C07281=1048.225,401.542,372.791,174.335,42.188,158.264
C07282=1048.234,401.788,372.747,174.343,42.195,158.266
C07283=1048.243,402.034,372.703,174.350,42.201,158.268
C07284=1048.252,402.280,372.659,174.359,42.208,158.271
C07285=1048.261,402.526,372.615,174.367,42.215,158.273
C07286=1048.270,402.772,372.571,174.375,42.222,158.275
C07287=1048.279,403.018,372.526,174.384,42.229,158.278
C07288=1048.288,403.264,372.482,174.391,42.236,158.280
C07289=1048.298,403.509,372.437,174.399,42.243,158.282
C07290=1048.311,403.897,372.367,174.413,42.254,158.286
C07291=1048.326,404.285,372.298,174.425,42.265,158.290
C07292=1048.340,404.673,372.227,174.439,42.276,158.294
C07293=1048.354,405.061,372.157,174.452,42.288,158.297
C07294=1048.363,405.308,372.113,174.461,42.295,158.300
C07295=1048.372,405.553,372.068,174.468,42.302,158.302
C07296=1048.381,405.799,372.022,174.478,42.309,158.305
C07297=1048.390,406.044,371.979,174.485,42.316,158.307
C07298=1048.399,406.290,371.933,174.495,42.324,158.310
C07299=1048.409,406.536,371.889,174.502,42.331,158.312
C07300=1048.417,406.782,371.844,174.511,42.338,158.314
C07301=1048.427,407.028,371.799,174.519,42.345,158.317
C07302=1048.436,407.274,371.754,174.528,42.353,158.319
C07303=1048.446,407.520,371.709,174.537,42.360,158.322
C07304=1048.455,407.765,371.664,174.545,42.367,158.324
C07305=1048.464,408.011,371.619,174.555,42.374,158.327
C07306=1048.473,408.257,371.574,174.563,42.382,158.329
C07307=1048.483,408.502,371.529,174.572,42.389,158.332
C07308=1048.492,408.748,371.483,174.580,42.397,158.334
C07309=1048.502,408.994,371.439,174.589,42.404,158.337
C07310=1048.511,409.239,371.393,174.598,42.412,158.339
C07311=1048.520,409.485,371.348,174.606,42.419,158.342
C07312=1048.529,409.731,371.303,174.615,42.427,158.344
C07313=1048.539,409.976,371.258,174.625,42.434,158.347
C07314=1048.548,410.222,371.213,174.633,42.442,158.350
C07315=1048.557,410.468,371.167,174.642,42.449,158.352
C07316=1048.567,410.714,371.122,174.651,42.456,158.355
C07317=1048.577,410.959,371.076,174.660,42.464,158.357
C07318=1048.586,411.205,371.031,174.669,42.472,158.360
C07319=1048.595,411.451,370.986,174.678,42.479,158.362
C07320=1048.606,411.696,370.940,174.687,42.487,158.365
C07321=1048.615,411.942,370.894,174.696,42.495,158.368
C07322=1048.624,412.187,370.848,174.705,42.502,158.370
C07323=1048.635,412.433,370.803,174.715,42.510,158.373
C07324=1048.643,412.679,370.758,174.724,42.518,158.376
C07325=1048.653,412.925,370.712,174.732,42.526,158.378
C07326=1048.663,413.170,370.665,174.742,42.534,158.381
C07327=1048.672,413.416,370.620,174.751,42.541,158.384
C07328=1048.682,413.662,370.574,174.761,42.549,158.387
C07329=1048.692,413.907,370.528,174.770,42.557,158.389
C07330=1048.701,414.152,370.481,174.779,42.565,158.392
C07331=1048.711,414.398,370.435,174.789,42.573,158.395
C07332=1048.720,414.643,370.389,174.798,42.581,158.397
C07333=1048.730,414.889,370.342,174.807,42.589,158.400
C07334=1048.739,415.134,370.296,174.817,42.597,158.403
C07335=1048.749,415.380,370.250,174.826,42.604,158.406
C07336=1048.758,415.626,370.204,174.836,42.613,158.409
C07337=1048.769,415.871,370.158,174.845,42.621,158.411
C07338=1048.778,416.116,370.111,174.855,42.629,158.414
C07339=1048.788,416.362,370.065,174.864,42.637,158.417
C07340=1048.797,416.607,370.019,174.874,42.645,158.420
C07341=1048.808,416.853,369.972,174.883,42.653,158.423
C07342=1048.817,417.099,369.925,174.893,42.662,158.425
C07343=1048.827,417.344,369.879,174.903,42.669,158.428
C07344=1048.837,417.589,369.832,174.913,42.678,158.431
C07345=1048.847,417.835,369.785,174.923,42.686,158.434
C07346=1048.862,418.230,369.710,174.939,42.699,158.439
C07347=1048.879,418.625,369.635,174.954,42.712,158.443
C07348=1048.895,419.020,369.559,174.970,42.726,158.448
C07349=1048.911,419.415,369.483,174.986,42.740,158.453
C07350=1048.921,419.660,369.437,174.996,42.748,158.456
C07351=1048.930,419.906,369.389,175.007,42.756,158.459
C07352=1048.940,420.152,369.342,175.017,42.765,158.462
C07353=1048.950,420.397,369.295,175.026,42.774,158.465
C07354=1048.960,420.642,369.248,175.037,42.782,158.468
C07355=1048.971,420.887,369.201,175.047,42.791,158.471
C07356=1048.980,421.133,369.153,175.058,42.799,158.474
C07357=1048.990,421.378,369.106,175.068,42.808,158.477
C07358=1049.001,421.623,369.058,175.078,42.816,158.480
C07359=1049.011,421.868,369.010,175.088,42.825,158.483
C07360=1049.020,422.114,368.963,175.098,42.834,158.486
C07361=1049.031,422.359,368.915,175.109,42.842,158.489
C07362=1049.041,422.604,368.868,175.119,42.851,158.492
C07363=1049.051,422.849,368.820,175.130,42.860,158.495
C07364=1049.061,423.094,368.773,175.141,42.868,158.499
C07365=1049.071,423.339,368.725,175.151,42.878,158.502
C07366=1049.082,423.585,368.677,175.162,42.886,158.505
C07367=1049.093,423.830,368.629,175.172,42.895,158.508
C07368=1049.103,424.075,368.582,175.183,42.904,158.511
C07369=1049.112,424.320,368.533,175.194,42.913,158.514
C07370=1049.123,424.566,368.486,175.204,42.922,158.518
C07371=1049.134,424.811,368.438,175.215,42.931,158.521
C07372=1049.144,425.056,368.389,175.226,42.939,158.524
C07373=1049.154,425.302,368.342,175.236,42.949,158.527
C07374=1049.165,425.546,368.294,175.247,42.957,158.530
C07375=1049.175,425.792,368.245,175.259,42.966,158.534
C07376=1049.186,426.037,368.197,175.270,42.976,158.537
C07377=1049.195,426.282,368.148,175.280,42.985,158.540
C07378=1049.207,426.527,368.100,175.291,42.994,158.544
C07379=1049.216,426.772,368.052,175.303,43.003,158.547
C07380=1049.227,427.017,368.003,175.314,43.012,158.550
C07381=1049.237,427.262,367.954,175.325,43.021,158.554
C07382=1049.249,427.507,367.906,175.336,43.031,158.557
C07383=1049.258,427.752,367.857,175.348,43.040,158.560
C07384=1049.269,427.997,367.809,175.359,43.049,158.564
C07385=1049.279,428.242,367.760,175.369,43.059,158.567
C07386=1049.291,428.487,367.711,175.381,43.068,158.571
C07387=1049.301,428.732,367.662,175.392,43.078,158.574
C07388=1049.311,428.977,367.613,175.403,43.087,158.577
C07389=1049.322,429.222,367.564,175.416,43.096,158.581
C07390=1049.332,429.467,367.516,175.427,43.106,158.584
C07391=1049.344,429.712,367.467,175.439,43.116,158.588
C07392=1049.354,429.957,367.417,175.450,43.125,158.591
C07393=1049.365,430.202,367.367,175.462,43.135,158.595
C07394=1049.375,430.447,367.319,175.473,43.144,158.599
C07395=1049.385,430.692,367.269,175.485,43.154,158.602
C07396=1049.397,430.937,367.220,175.496,43.163,158.606
C07397=1049.407,431.182,367.171,175.508,43.173,158.609
C07398=1049.417,431.426,367.121,175.521,43.183,158.613
C07399=1049.428,431.671,367.072,175.532,43.193,158.616
C07400=1049.440,431.915,367.022,175.544,43.203,158.620
C07401=1049.451,432.160,366.973,175.557,43.212,158.624
C07402=1049.459,432.370,366.930,175.567,43.221,158.627
C07403=1049.469,432.579,366.888,175.577,43.229,158.630
C07404=1049.478,432.788,366.845,175.587,43.237,158.633
C07405=1049.487,432.997,366.803,175.598,43.246,158.636
C07406=1049.498,433.207,366.760,175.608,43.254,158.639
C07407=1049.507,433.416,366.717,175.618,43.263,158.642
C07408=1049.516,433.625,366.675,175.629,43.271,158.646
C07409=1049.525,433.834,366.632,175.639,43.280,158.649
C07410=1049.536,434.079,366.583,175.651,43.290,158.653
C07411=1049.547,434.323,366.533,175.664,43.300,158.656
C07412=1049.559,434.569,366.482,175.676,43.310,158.660
C07413=1049.570,434.813,366.432,175.689,43.320,158.664
C07414=1049.581,435.058,366.382,175.702,43.330,158.668
C07415=1049.592,435.302,366.332,175.714,43.341,158.672
C07416=1049.604,435.547,366.282,175.726,43.351,158.675
C07417=1049.615,435.792,366.231,175.739,43.361,158.679
C07418=1049.626,436.036,366.181,175.752,43.371,158.683
C07419=1049.637,436.281,366.130,175.764,43.381,158.687
C07420=1049.648,436.526,366.080,175.778,43.391,158.691
C07421=1049.659,436.770,366.030,175.790,43.402,158.695
C07422=1049.671,437.015,365.979,175.803,43.412,158.699
C07423=1049.682,437.259,365.928,175.816,43.423,158.703
C07424=1049.694,437.504,365.877,175.829,43.433,158.707
C07425=1049.705,437.749,365.827,175.841,43.444,158.711
C07426=1049.717,437.993,365.776,175.855,43.455,158.715
C07427=1049.728,438.238,365.725,175.868,43.465,158.719
C07428=1049.740,438.482,365.674,175.881,43.476,158.723
C07429=1049.750,438.727,365.624,175.894,43.486,158.727
C07430=1049.762,438.971,365.572,175.908,43.497,158.731
C07431=1049.774,439.216,365.520,175.921,43.508,158.735
C07432=1049.785,439.460,365.469,175.935,43.518,158.739
C07433=1049.797,439.704,365.418,175.948,43.529,158.743
C07434=1049.808,439.949,365.367,175.961,43.540,158.747
C07435=1049.820,440.193,365.316,175.975,43.551,158.751
C07436=1049.831,440.438,365.264,175.988,43.562,158.756
C07437=1049.843,440.682,365.212,176.002,43.573,158.760
C07438=1049.855,440.926,365.160,176.016,43.583,158.764
C07439=1049.866,441.170,365.109,176.030,43.594,158.768
C07440=1049.878,441.415,365.058,176.043,43.605,158.772
C07441=1049.890,441.659,365.007,176.057,43.616,158.777
C07442=1049.901,441.903,364.954,176.072,43.627,158.781
C07443=1049.913,442.148,364.902,176.085,43.639,158.785
C07444=1049.925,442.392,364.850,176.099,43.650,158.790
C07445=1049.936,442.637,364.798,176.114,43.661,158.794
C07446=1049.949,442.880,364.746,176.128,43.672,158.798
C07447=1049.961,443.124,364.694,176.141,43.683,158.803
C07448=1049.973,443.369,364.643,176.156,43.695,158.807
C07449=1049.984,443.613,364.590,176.170,43.706,158.812
C07450=1049.996,443.857,364.538,176.185,43.717,158.816
C07451=1050.009,444.101,364.486,176.199,43.729,158.821
C07452=1050.020,444.345,364.433,176.214,43.740,158.825
C07453=1050.033,444.590,364.381,176.229,43.752,158.830
C07454=1050.045,444.834,364.328,176.243,43.763,158.834
C07455=1050.056,445.078,364.276,176.258,43.775,158.839
C07456=1050.069,445.322,364.223,176.273,43.786,158.843
C07457=1050.081,445.566,364.171,176.287,43.798,158.848
C07458=1050.093,445.809,364.119,176.302,43.809,158.852
C07459=1050.106,446.052,364.066,176.317,43.821,158.857
C07460=1050.119,446.296,364.014,176.332,43.832,158.862
C07461=1050.132,446.540,363.962,176.347,43.843,158.866
C07462=1050.148,446.805,363.907,176.364,43.856,158.871
C07463=1050.165,447.073,363.851,176.380,43.868,158.876
C07464=1050.182,447.340,363.797,176.396,43.879,158.881
C07465=1050.201,447.608,363.743,176.414,43.891,158.886
C07466=1050.219,447.852,363.694,176.430,43.901,158.890
C07467=1050.237,448.096,363.647,176.444,43.912,158.894
C07468=1050.255,448.341,363.599,176.460,43.922,158.899
C07469=1050.275,448.586,363.552,176.476,43.932,158.903
C07470=1050.296,448.830,363.505,176.492,43.942,158.907
C07471=1050.317,449.075,363.459,176.508,43.951,158.911
C07472=1050.338,449.321,363.414,176.523,43.961,158.916
C07473=1050.361,449.566,363.369,176.540,43.971,158.920
C07474=1050.384,449.811,363.325,176.556,43.980,158.924
C07475=1050.408,450.056,363.281,176.572,43.989,158.928
C07476=1050.432,450.302,363.238,176.588,43.998,158.932
C07477=1050.458,450.546,363.195,176.605,44.007,158.936
C07478=1050.144,450.574,362.895,176.604,44.099,158.963
C07479=1050.118,450.329,362.938,176.588,44.090,158.959
C07480=1050.094,450.083,362.981,176.572,44.081,158.955
C07481=1050.070,449.838,363.025,176.556,44.073,158.951
C07482=1050.046,449.593,363.069,176.539,44.064,158.947
C07483=1050.024,449.348,363.113,176.523,44.054,158.942
C07484=1050.002,449.103,363.159,176.507,44.044,158.938
C07485=1049.981,448.858,363.205,176.492,44.034,158.934
C07486=1049.960,448.613,363.251,176.475,44.025,158.930
C07487=1049.941,448.368,363.298,176.460,44.015,158.925
C07488=1049.921,448.124,363.346,176.444,44.005,158.921
C07489=1049.903,447.880,363.393,176.428,43.995,158.917
C07490=1049.886,447.636,363.442,176.412,43.985,158.912
C07491=1049.868,447.386,363.493,176.397,43.973,158.908
C07492=1049.851,447.137,363.543,176.381,43.963,158.903
C07493=1049.836,446.888,363.594,176.365,43.952,158.899
C07494=1049.821,446.639,363.646,176.350,43.940,158.894
C07495=1049.806,446.395,363.697,176.335,43.929,158.890
C07496=1049.792,446.151,363.749,176.320,43.918,158.885
C07497=1049.779,445.908,363.801,176.305,43.907,158.881
C07498=1049.767,445.666,363.853,176.290,43.895,158.876
C07499=1049.755,445.422,363.906,176.275,43.884,158.871
C07500=1049.743,445.177,363.959,176.260,43.872,158.867
C07501=1049.730,444.933,364.011,176.246,43.861,158.862
C07502=1049.719,444.690,364.064,176.231,43.850,158.858
C07503=1049.706,444.446,364.116,176.216,43.838,158.853
C07504=1049.694,444.201,364.169,176.202,43.826,158.849
C07505=1049.682,443.957,364.221,176.187,43.816,158.844
C07506=1049.670,443.713,364.274,176.173,43.804,158.840
C07507=1049.658,443.469,364.325,176.158,43.793,158.835
C07508=1049.647,443.224,364.378,176.144,43.782,158.831
C07509=1049.635,442.980,364.430,176.129,43.770,158.826
C07510=1049.622,442.737,364.482,176.115,43.759,158.822
C07511=1049.611,442.492,364.534,176.101,43.748,158.818
C07512=1049.599,442.248,364.586,176.087,43.737,158.813
C07513=1049.587,442.003,364.637,176.072,43.726,158.809
C07514=1049.575,441.759,364.690,176.059,43.715,158.805
C07515=1049.564,441.515,364.742,176.045,43.704,158.800
C07516=1049.552,441.270,364.793,176.030,43.693,158.796
C07517=1049.540,441.026,364.845,176.017,43.682,158.792
C07518=1049.528,440.782,364.896,176.003,43.672,158.788
C07519=1049.516,440.537,364.948,175.989,43.660,158.783
C07520=1049.504,440.293,364.999,175.976,43.650,158.779
C07521=1049.494,440.049,365.051,175.962,43.639,158.775
C07522=1049.482,439.804,365.102,175.948,43.628,158.771
C07523=1049.470,439.560,365.154,175.935,43.618,158.767
C07524=1049.458,439.316,365.205,175.921,43.607,158.763
C07525=1049.447,439.071,365.256,175.908,43.596,158.759
C07526=1049.435,438.826,365.307,175.894,43.585,158.754
C07527=1049.424,438.582,365.358,175.881,43.575,158.750
C07528=1049.413,438.337,365.410,175.868,43.564,158.746
C07529=1049.401,438.092,365.461,175.855,43.554,158.742
C07530=1049.390,437.849,365.512,175.841,43.543,158.738
C07531=1049.378,437.603,365.562,175.829,43.533,158.734
C07532=1049.367,437.360,365.613,175.816,43.522,158.730
C07533=1049.355,437.114,365.664,175.803,43.512,158.726
C07534=1049.344,436.870,365.714,175.789,43.502,158.722
C07535=1049.333,436.626,365.765,175.776,43.492,158.718
C07536=1049.322,436.381,365.816,175.764,43.481,158.715
C07537=1049.311,436.137,365.866,175.751,43.471,158.711
C07538=1049.299,435.892,365.917,175.738,43.460,158.707
C07539=1049.287,435.647,365.967,175.725,43.451,158.703
C07540=1049.276,435.403,366.017,175.713,43.440,158.699
C07541=1049.265,435.158,366.068,175.700,43.430,158.695
C07542=1049.254,434.913,366.117,175.687,43.420,158.691
C07543=1049.243,434.668,366.168,175.675,43.410,158.688
C07544=1049.231,434.424,366.218,175.662,43.400,158.684
C07545=1049.220,434.180,366.268,175.650,43.390,158.680
C07546=1049.209,433.934,366.318,175.637,43.380,158.676
C07547=1049.200,433.724,366.361,175.627,43.372,158.673
C07548=1049.190,433.514,366.404,175.616,43.363,158.670
C07549=1049.180,433.304,366.446,175.606,43.355,158.667
C07550=1049.171,433.094,366.489,175.596,43.346,158.663
C07551=1049.161,432.884,366.532,175.585,43.338,158.660
C07552=1049.152,432.673,366.575,175.574,43.329,158.657
C07553=1049.143,432.463,366.618,175.563,43.321,158.654
C07554=1049.134,432.253,366.660,175.553,43.313,158.651
C07555=1049.123,432.008,366.710,175.542,43.302,158.647
C07556=1049.112,431.764,366.759,175.530,43.293,158.644
C07557=1049.101,431.519,366.809,175.517,43.283,158.640
C07558=1049.090,431.274,366.859,175.506,43.273,158.636
C07559=1049.080,431.029,366.908,175.494,43.264,158.633
C07560=1049.068,430.784,366.957,175.482,43.254,158.629
C07561=1049.058,430.539,367.007,175.470,43.244,158.626
C07562=1049.048,430.294,367.056,175.458,43.235,158.622
C07563=1049.037,430.049,367.106,175.447,43.225,158.618
C07564=1049.026,429.804,367.154,175.435,43.216,158.615
C07565=1049.015,429.559,367.204,175.424,43.207,158.612
C07566=1049.005,429.315,367.253,175.412,43.197,158.608
C07567=1048.994,429.070,367.302,175.401,43.187,158.605
C07568=1048.983,428.824,367.351,175.389,43.178,158.601
C07569=1048.973,428.578,367.400,175.377,43.169,158.598
C07570=1048.962,428.334,367.448,175.366,43.160,158.594
C07571=1048.952,428.089,367.497,175.354,43.150,158.591
C07572=1048.941,427.845,367.546,175.343,43.141,158.587
C07573=1048.931,427.599,367.595,175.332,43.132,158.584
C07574=1048.920,427.354,367.643,175.321,43.123,158.581
C07575=1048.909,427.109,367.692,175.310,43.113,158.577
C07576=1048.898,426.864,367.741,175.298,43.104,158.574
C07577=1048.889,426.619,367.789,175.287,43.095,158.571
C07578=1048.878,426.374,367.837,175.276,43.086,158.567
C07579=1048.868,426.129,367.886,175.265,43.077,158.564
C07580=1048.857,425.884,367.934,175.254,43.068,158.561
C07581=1048.847,425.638,367.983,175.243,43.059,158.557
C07582=1048.836,425.394,368.031,175.232,43.050,158.554
C07583=1048.826,425.149,368.079,175.221,43.041,158.551
C07584=1048.816,424.903,368.128,175.210,43.032,158.548
C07585=1048.805,424.658,368.175,175.200,43.023,158.545
C07586=1048.794,424.413,368.223,175.189,43.014,158.541
C07587=1048.785,424.168,368.272,175.178,43.005,158.538
C07588=1048.774,423.922,368.319,175.168,42.997,158.535
C07589=1048.764,423.678,368.367,175.157,42.988,158.532
C07590=1048.753,423.432,368.414,175.146,42.979,158.529
C07591=1048.743,423.187,368.463,175.135,42.970,158.525
C07592=1048.733,422.942,368.510,175.124,42.961,158.522
C07593=1048.723,422.697,368.558,175.114,42.953,158.519
C07594=1048.712,422.452,368.605,175.104,42.944,158.516
C07595=1048.703,422.206,368.653,175.093,42.936,158.513
C07596=1048.693,421.961,368.700,175.083,42.927,158.510
C07597=1048.682,421.716,368.748,175.072,42.918,158.507
C07598=1048.671,421.470,368.796,175.062,42.910,158.504
C07599=1048.661,421.225,368.843,175.052,42.901,158.501
C07600=1048.652,420.980,368.890,175.041,42.893,158.498
C07601=1048.642,420.735,368.938,175.031,42.884,158.495
C07602=1048.632,420.489,368.985,175.020,42.876,158.491
C07603=1048.622,420.244,369.032,175.011,42.867,158.489
C07604=1048.612,419.999,369.079,175.001,42.859,158.486
C07605=1048.602,419.753,369.127,174.990,42.850,158.482
C07606=1048.592,419.508,369.174,174.980,42.842,158.480
C07607=1048.576,419.111,369.250,174.964,42.828,158.475
C07608=1048.560,418.714,369.326,174.947,42.815,158.470
C07609=1048.544,418.317,369.402,174.931,42.801,158.465
C07610=1048.528,417.920,369.477,174.915,42.788,158.461
C07611=1048.517,417.674,369.524,174.906,42.780,158.458
C07612=1048.508,417.429,369.571,174.896,42.772,158.455
C07613=1048.498,417.183,369.617,174.886,42.764,158.452
C07614=1048.488,416.938,369.664,174.876,42.756,158.449
C07615=1048.478,416.692,369.711,174.866,42.748,158.446
C07616=1048.468,416.446,369.757,174.857,42.740,158.443
C07617=1048.459,416.202,369.804,174.847,42.731,158.441
C07618=1048.449,415.956,369.851,174.838,42.724,158.438
C07619=1048.440,415.711,369.897,174.828,42.715,158.435
C07620=1048.430,415.465,369.943,174.819,42.707,158.432
C07621=1048.419,415.219,369.989,174.809,42.700,158.429
C07622=1048.410,414.974,370.035,174.800,42.692,158.427
C07623=1048.400,414.728,370.082,174.790,42.684,158.424
C07624=1048.391,414.483,370.128,174.781,42.676,158.421
C07625=1048.381,414.238,370.174,174.771,42.668,158.418
C07626=1048.371,413.992,370.221,174.762,42.660,158.416
C07627=1048.362,413.746,370.267,174.753,42.652,158.413
C07628=1048.352,413.501,370.313,174.743,42.645,158.410
C07629=1048.343,413.255,370.359,174.734,42.637,158.407
C07630=1048.333,413.010,370.404,174.724,42.629,158.405
C07631=1048.323,412.764,370.451,174.715,42.621,158.402
C07632=1048.314,412.518,370.496,174.706,42.614,158.399
C07633=1048.304,412.272,370.543,174.696,42.606,158.397
C07634=1048.295,412.027,370.587,174.687,42.598,158.394
C07635=1048.285,411.781,370.634,174.679,42.590,158.391
C07636=1048.275,411.535,370.679,174.670,42.583,158.389
C07637=1048.266,411.289,370.724,174.660,42.575,158.386
C07638=1048.257,411.044,370.770,174.651,42.568,158.384
C07639=1048.247,410.799,370.815,174.642,42.560,158.381
C07640=1048.238,410.552,370.861,174.634,42.553,158.378
C07641=1048.228,410.307,370.906,174.625,42.545,158.376
C07642=1048.219,410.061,370.952,174.615,42.538,158.373
C07643=1048.209,409.816,370.997,174.606,42.530,158.371
C07644=1048.200,409.570,371.042,174.598,42.523,158.368
C07645=1048.190,409.325,371.087,174.589,42.515,158.365
C07646=1048.181,409.078,371.133,174.580,42.508,158.363
C07647=1048.171,408.833,371.178,174.570,42.500,158.360
C07648=1048.162,408.587,371.223,174.562,42.493,158.358
C07649=1048.152,408.341,371.268,174.553,42.486,158.355
C07650=1048.143,408.095,371.313,174.545,42.479,158.353
C07651=1048.134,407.850,371.359,174.536,42.471,158.350
C07652=1048.125,407.604,371.403,174.527,42.464,158.348
C07653=1048.116,407.358,371.449,174.519,42.457,158.345
C07654=1048.106,407.112,371.493,174.510,42.449,158.343
C07655=1048.097,406.866,371.538,174.502,42.442,158.341
C07656=1048.088,406.622,371.583,174.493,42.435,158.338
C07657=1048.079,406.376,371.628,174.484,42.428,158.336
C07658=1048.070,406.130,371.672,174.476,42.420,158.333
C07659=1048.061,405.884,371.718,174.467,42.414,158.331
C07660=1048.051,405.638,371.762,174.459,42.407,158.328
C07661=1048.042,405.392,371.807,174.450,42.399,158.326
C07662=1048.034,405.146,371.851,174.442,42.392,158.323
C07663=1048.019,404.757,371.922,174.428,42.381,158.320
C07664=1048.004,404.366,371.993,174.415,42.370,158.316
C07665=1047.990,403.976,372.064,174.402,42.359,158.312
C07666=1047.976,403.586,372.134,174.389,42.348,158.308
C07667=1047.967,403.341,372.178,174.380,42.341,158.306
C07668=1047.958,403.095,372.223,174.373,42.334,158.304
C07669=1047.948,402.849,372.267,174.364,42.327,158.301
C07670=1047.940,402.603,372.311,174.356,42.320,158.299
C07671=1047.931,402.357,372.355,174.348,42.313,158.297
C07672=1047.921,402.111,372.400,174.339,42.306,158.295
C07673=1047.913,401.865,372.443,174.331,42.299,158.292
C07674=1047.903,401.619,372.487,174.324,42.293,158.290
C07675=1047.894,401.374,372.531,174.315,42.286,158.288
C07676=1047.886,401.127,372.576,174.307,42.279,158.285
C07677=1047.877,400.882,372.620,174.299,42.272,158.283
C07678=1047.868,400.635,372.663,174.292,42.266,158.281
C07679=1047.859,400.389,372.707,174.283,42.259,158.279
C07680=1047.850,400.143,372.751,174.275,42.252,158.276
C07681=1047.841,399.898,372.795,174.267,42.246,158.274
C07682=1047.832,399.651,372.838,174.260,42.239,158.272
C07683=1047.823,399.406,372.882,174.251,42.232,158.270
C07684=1047.814,399.160,372.925,174.243,42.226,158.268
C07685=1047.805,398.914,372.969,174.236,42.219,158.265
C07686=1047.796,398.668,373.013,174.228,42.213,158.263
C07687=1047.788,398.422,373.056,174.220,42.206,158.261
C07688=1047.778,398.176,373.100,174.213,42.199,158.259
C07689=1047.770,397.930,373.143,174.204,42.193,158.257
C07690=1047.761,397.684,373.186,174.197,42.187,158.254
C07691=1047.752,397.438,373.230,174.189,42.180,158.252
C07692=1047.743,397.192,373.273,174.181,42.173,158.250
C07693=1047.735,396.946,373.317,174.174,42.167,158.248
C07694=1047.726,396.700,373.360,174.166,42.160,158.246
C07695=1047.718,396.454,373.403,174.159,42.154,158.244
C07696=1047.708,396.207,373.446,174.151,42.148,158.242
C07697=1047.700,395.962,373.490,174.143,42.141,158.239
C07698=1047.691,395.716,373.533,174.135,42.135,158.237
C07699=1047.683,395.470,373.576,174.127,42.129,158.235
C07700=1047.673,395.224,373.618,174.120,42.122,158.233
C07701=1047.665,394.978,373.661,174.112,42.116,158.231
C07702=1047.656,394.732,373.704,174.105,42.110,158.229
C07703=1047.647,394.485,373.748,174.097,42.104,158.227
C07704=1047.639,394.239,373.791,174.090,42.097,158.225
C07705=1047.630,393.993,373.833,174.082,42.091,158.223
C07706=1047.621,393.747,373.876,174.075,42.085,158.221
C07707=1047.613,393.501,373.919,174.067,42.078,158.219
C07708=1047.604,393.255,373.962,174.060,42.072,158.217
C07709=1047.596,393.009,374.005,174.052,42.066,158.215
C07710=1047.587,392.763,374.047,174.045,42.060,158.213
C07711=1047.578,392.517,374.090,174.039,42.054,158.211
C07712=1047.571,392.271,374.132,174.031,42.047,158.209
C07713=1047.562,392.025,374.175,174.024,42.041,158.207
C07714=1047.553,391.779,374.218,174.016,42.035,158.205
C07715=1047.545,391.532,374.260,174.009,42.029,158.203
C07716=1047.536,391.286,374.303,174.001,42.023,158.201
C07717=1047.527,391.040,374.345,173.994,42.017,158.199
C07718=1047.519,390.794,374.388,173.987,42.011,158.197
C07719=1047.506,390.422,374.451,173.976,42.002,158.194
C07720=1047.493,390.051,374.515,173.966,41.993,158.191
C07721=1047.480,389.680,374.578,173.954,41.984,158.188
C07722=1047.468,389.309,374.642,173.944,41.975,158.185
C07723=1047.459,389.062,374.684,173.936,41.970,158.183
C07724=1047.451,388.816,374.727,173.930,41.963,158.181
C07725=1047.441,388.570,374.769,173.923,41.957,158.179
C07726=1047.434,388.324,374.811,173.916,41.952,158.177
C07727=1047.425,388.078,374.853,173.908,41.946,158.175
C07728=1047.416,387.831,374.894,173.901,41.940,158.174
C07729=1047.408,387.584,374.937,173.895,41.935,158.172
C07730=1047.399,387.339,374.978,173.888,41.928,158.170
C07731=1047.391,387.092,375.020,173.880,41.923,158.168
C07732=1047.382,386.846,375.062,173.873,41.917,158.166
C07733=1047.374,386.600,375.103,173.867,41.911,158.164
C07734=1047.365,386.354,375.145,173.860,41.906,158.162
C07735=1047.357,386.106,375.187,173.853,41.900,158.160
C07736=1047.349,385.861,375.228,173.845,41.894,158.159
C07737=1047.340,385.614,375.270,173.839,41.888,158.157
C07738=1047.332,385.368,375.312,173.832,41.883,158.155
C07739=1047.323,385.122,375.353,173.825,41.877,158.153
C07740=1047.315,384.876,375.394,173.819,41.872,158.151
C07741=1047.307,384.629,375.436,173.811,41.866,158.149
C07742=1047.298,384.383,375.478,173.805,41.860,158.148
C07743=1047.290,384.136,375.519,173.798,41.855,158.146
C07744=1047.282,383.890,375.561,173.791,41.849,158.144
C07745=1047.274,383.644,375.602,173.785,41.844,158.142
C07746=1047.266,383.398,375.643,173.778,41.838,158.140
C07747=1047.257,383.151,375.685,173.771,41.832,158.139
C07748=1047.249,382.905,375.726,173.764,41.827,158.137
C07749=1047.240,382.659,375.768,173.757,41.821,158.135
C07750=1047.232,382.412,375.808,173.751,41.816,158.133
C07751=1047.225,382.165,375.850,173.744,41.810,158.132
C07752=1047.216,381.919,375.891,173.738,41.805,158.130
C07753=1047.208,381.673,375.932,173.731,41.799,158.128
C07754=1047.200,381.426,375.974,173.725,41.794,158.126
C07755=1047.192,381.180,376.015,173.718,41.789,158.125
C07756=1047.184,380.934,376.055,173.712,41.783,158.123
C07757=1047.175,380.687,376.096,173.705,41.778,158.121
C07758=1047.168,380.441,376.138,173.699,41.772,158.119
C07759=1047.160,380.195,376.179,173.692,41.766,158.118
C07760=1047.152,379.948,376.220,173.686,41.761,158.116
C07761=1047.144,379.701,376.261,173.679,41.756,158.114
C07762=1047.136,379.455,376.302,173.673,41.751,158.112
C07763=1047.128,379.208,376.343,173.666,41.745,158.111
C07764=1047.120,378.962,376.383,173.660,41.740,158.109
C07765=1047.111,378.715,376.424,173.653,41.735,158.107
C07766=1047.103,378.469,376.465,173.647,41.730,158.106
C07767=1047.094,378.212,376.508,173.640,41.724,158.104
C07768=1047.086,377.954,376.550,173.634,41.718,158.102
C07769=1047.077,377.698,376.592,173.626,41.713,158.100
C07770=1047.069,377.440,376.634,173.620,41.708,158.099
C07771=1047.061,377.194,376.675,173.614,41.703,158.097
C07772=1047.053,376.947,376.715,173.608,41.697,158.096
C07773=1047.044,376.700,376.756,173.601,41.692,158.094
C07774=1047.036,376.453,376.796,173.595,41.687,158.092
C07775=1047.025,376.126,376.849,173.586,41.680,158.090
C07776=1047.015,375.798,376.903,173.578,41.673,158.088
C07777=1047.004,375.472,376.957,173.569,41.667,158.086
C07778=1046.994,375.144,377.011,173.562,41.659,158.083
C07779=1046.986,374.897,377.050,173.555,41.654,158.082
C07780=1046.978,374.651,377.091,173.549,41.649,158.080
C07781=1046.970,374.404,377.131,173.543,41.645,158.079
C07782=1046.962,374.158,377.171,173.536,41.640,158.077
C07783=1046.954,373.911,377.211,173.530,41.634,158.076
C07784=1046.946,373.665,377.252,173.524,41.629,158.074
C07785=1046.938,373.418,377.292,173.518,41.624,158.072
C07786=1046.931,373.171,377.332,173.512,41.620,158.071
C07787=1046.923,372.925,377.372,173.506,41.614,158.069
C07788=1046.915,372.678,377.412,173.500,41.609,158.068
C07789=1046.906,372.431,377.452,173.493,41.604,158.066
C07790=1046.899,372.186,377.492,173.487,41.599,158.064
C07791=1046.891,371.939,377.532,173.482,41.594,158.063
C07792=1046.884,371.692,377.572,173.476,41.589,158.061
C07793=1046.876,371.445,377.612,173.470,41.584,158.060
C07794=1046.868,371.198,377.652,173.463,41.579,158.058
C07795=1046.860,370.951,377.692,173.457,41.575,158.057
C07796=1046.852,370.705,377.731,173.452,41.570,158.055
C07797=1046.844,370.458,377.771,173.446,41.565,158.054
C07798=1046.836,370.211,377.810,173.439,41.560,158.052
C07799=1046.829,369.965,377.850,173.433,41.555,158.051
C07800=1046.821,369.718,377.890,173.428,41.551,158.049
C07801=1046.812,369.471,377.929,173.422,41.546,158.048
C07802=1046.805,369.224,377.969,173.416,41.541,158.046
C07803=1046.796,368.978,378.008,173.409,41.536,158.045
C07804=1046.789,368.732,378.048,173.404,41.532,158.043
C07805=1046.781,368.485,378.087,173.398,41.527,158.042
C07806=1046.773,368.237,378.126,173.392,41.522,158.040
C07807=1046.765,367.991,378.166,173.386,41.517,158.039
C07808=1046.758,367.745,378.205,173.381,41.512,158.037
C07809=1046.750,367.498,378.245,173.375,41.508,158.036
C07810=1046.742,367.251,378.284,173.369,41.503,158.034
C07811=1046.734,367.004,378.324,173.363,41.499,158.033
C07812=1046.726,366.758,378.363,173.357,41.494,158.031
C07813=1046.719,366.510,378.402,173.351,41.489,158.030
C07814=1046.710,366.264,378.441,173.346,41.484,158.028
C07815=1046.704,366.017,378.480,173.340,41.479,158.027
C07816=1046.695,365.770,378.519,173.334,41.475,158.025
C07817=1046.688,365.524,378.559,173.328,41.470,158.024
C07818=1046.680,365.277,378.597,173.323,41.466,158.023
C07819=1046.672,365.030,378.637,173.317,41.461,158.021
C07820=1046.665,364.783,378.676,173.312,41.457,158.020
C07821=1046.657,364.536,378.715,173.306,41.452,158.018
C07822=1046.650,364.290,378.754,173.300,41.447,158.017
C07823=1046.642,364.042,378.793,173.295,41.443,158.015
C07824=1046.635,363.796,378.832,173.289,41.438,158.014
C07825=1046.627,363.549,378.871,173.283,41.433,158.013
C07826=1046.620,363.302,378.910,173.278,41.429,158.011
C07827=1046.611,363.056,378.949,173.272,41.424,158.010
C07828=1046.605,362.809,378.988,173.267,41.420,158.008
C07829=1046.596,362.562,379.027,173.261,41.415,158.007
C07830=1046.589,362.315,379.065,173.255,41.411,158.006
C07831=1046.578,361.996,379.115,173.248,41.405,158.004
C07832=1046.568,361.677,379.165,173.240,41.399,158.002
C07833=1046.559,361.358,379.215,173.233,41.393,158.000
C07834=1046.549,361.040,379.265,173.226,41.388,157.998
C07835=1046.541,360.792,379.304,173.221,41.384,157.997
C07836=1046.534,360.546,379.342,173.215,41.379,157.996
C07837=1046.526,360.299,379.380,173.210,41.375,157.994
C07838=1046.518,360.052,379.419,173.204,41.370,157.993
C07839=1046.511,359.805,379.457,173.199,41.366,157.992
C07840=1046.504,359.557,379.496,173.194,41.362,157.990
C07841=1046.496,359.311,379.534,173.188,41.357,157.989
C07842=1046.488,359.064,379.572,173.183,41.353,157.988
C07843=1046.480,358.817,379.611,173.177,41.348,157.986
C07844=1046.473,358.570,379.649,173.172,41.344,157.985
C07845=1046.466,358.324,379.688,173.166,41.340,157.984
C07846=1046.458,358.076,379.726,173.161,41.336,157.982
C07847=1046.451,357.829,379.764,173.155,41.331,157.981
C07848=1046.443,357.583,379.802,173.151,41.327,157.980
C07849=1046.435,357.335,379.840,173.145,41.323,157.978
C07850=1046.428,357.088,379.878,173.140,41.319,157.977
C07851=1046.420,356.842,379.917,173.134,41.314,157.976
C07852=1046.413,356.595,379.954,173.129,41.310,157.974
C07853=1046.405,356.348,379.993,173.123,41.306,157.973
C07854=1046.397,356.100,380.030,173.118,41.302,157.972
C07855=1046.390,355.854,380.069,173.113,41.297,157.971
C07856=1046.383,355.607,380.106,173.108,41.293,157.969
C07857=1046.374,355.360,380.145,173.102,41.289,157.968
C07858=1046.367,355.112,380.182,173.097,41.285,157.967
C07859=1046.360,354.866,380.221,173.092,41.281,157.966
C07860=1046.352,354.619,380.258,173.086,41.277,157.964
C07861=1046.345,354.372,380.296,173.082,41.272,157.963
C07862=1046.337,354.124,380.334,173.076,41.268,157.962
C07863=1046.330,353.877,380.372,173.071,41.264,157.960
C07864=1046.322,353.631,380.410,173.065,41.260,157.959
C07865=1046.315,353.384,380.447,173.061,41.256,157.958
C07866=1046.308,353.137,380.485,173.055,41.252,157.957
C07867=1046.300,352.889,380.523,173.050,41.247,157.955
C07868=1046.293,352.643,380.561,173.045,41.243,157.954
C07869=1046.286,352.396,380.598,173.040,41.240,157.953
C07870=1046.278,352.148,380.636,173.035,41.235,157.952
C07871=1046.271,351.901,380.674,173.029,41.231,157.950
C07872=1046.263,351.654,380.711,173.024,41.227,157.949
C07873=1046.256,351.406,380.749,173.020,41.223,157.948
C07874=1046.249,351.160,380.787,173.014,41.219,157.947
C07875=1046.241,350.913,380.824,173.009,41.215,157.945
C07876=1046.233,350.666,380.861,173.004,41.211,157.944
C07877=1046.226,350.419,380.899,172.999,41.207,157.943
C07878=1046.219,350.172,380.937,172.994,41.203,157.942
C07879=1046.212,349.925,380.974,172.989,41.199,157.941
C07880=1046.204,349.677,381.012,172.984,41.195,157.939
C07881=1046.197,349.430,381.048,172.979,41.191,157.938
C07882=1046.189,349.183,381.085,172.973,41.187,157.937
C07883=1046.182,348.936,381.123,172.969,41.183,157.936
C07884=1046.174,348.689,381.160,172.963,41.179,157.935
C07885=1046.167,348.442,381.197,172.958,41.176,157.933
C07886=1046.160,348.195,381.235,172.954,41.171,157.932
C07887=1046.151,347.882,381.282,172.947,41.167,157.931
C07888=1046.141,347.569,381.329,172.941,41.161,157.929
C07889=1046.132,347.255,381.375,172.935,41.157,157.928
C07890=1046.123,346.941,381.422,172.928,41.151,157.926
C07891=1046.116,346.694,381.460,172.924,41.148,157.925
C07892=1046.108,346.447,381.497,172.919,41.144,157.924
C07893=1046.101,346.200,381.533,172.914,41.140,157.923
C07894=1046.094,345.953,381.571,172.909,41.136,157.922
C07895=1046.086,345.706,381.607,172.904,41.133,157.920
C07896=1046.079,345.459,381.645,172.899,41.128,157.919
C07897=1046.071,345.212,381.681,172.894,41.125,157.918
C07898=1046.064,344.964,381.718,172.890,41.121,157.917
C07899=1046.057,344.718,381.755,172.884,41.117,157.916
C07900=1046.050,344.470,381.792,172.879,41.113,157.915
C07901=1046.043,344.223,381.829,172.875,41.110,157.913
C07902=1046.035,343.975,381.865,172.870,41.106,157.912
C07903=1046.029,343.728,381.902,172.865,41.102,157.911
C07904=1046.021,343.482,381.939,172.860,41.098,157.910
C07905=1046.014,343.234,381.976,172.856,41.094,157.909
C07906=1046.006,342.986,382.012,172.850,41.091,157.908
C07907=1045.999,342.740,382.049,172.846,41.087,157.907
C07908=1045.992,342.492,382.086,172.841,41.083,157.906
C07909=1045.985,342.245,382.122,172.837,41.079,157.904
C07910=1045.977,341.998,382.160,172.831,41.075,157.903
C07911=1045.970,341.751,382.195,172.827,41.072,157.902
C07912=1045.963,341.503,382.232,172.822,41.068,157.901
C07913=1045.956,341.256,382.268,172.817,41.064,157.900
C07914=1045.949,341.009,382.304,172.812,41.061,157.899
C07915=1045.941,340.761,382.340,172.807,41.057,157.898
C07916=1045.934,340.514,382.378,172.803,41.053,157.897
C07917=1045.927,340.268,382.414,172.798,41.050,157.895
C07918=1045.919,340.020,382.450,172.793,41.046,157.894
C07919=1045.912,339.772,382.487,172.789,41.043,157.893
C07920=1045.905,339.526,382.523,172.784,41.039,157.892
C07921=1045.897,339.278,382.559,172.780,41.036,157.891
C07922=1045.891,339.031,382.595,172.775,41.032,157.890
C07923=1045.883,338.784,382.632,172.770,41.028,157.889
C07924=1045.876,338.536,382.668,172.765,41.025,157.888
C07925=1045.869,338.290,382.704,172.761,41.021,157.887
C07926=1045.862,338.041,382.740,172.756,41.017,157.886
C07927=1045.855,337.794,382.776,172.752,41.014,157.885
C07928=1045.847,337.547,382.812,172.747,41.010,157.884
C07929=1045.841,337.300,382.848,172.742,41.007,157.883
C07930=1045.833,337.052,382.885,172.738,41.003,157.881
C07931=1045.826,336.806,382.920,172.733,40.999,157.880
C07932=1045.819,336.558,382.957,172.729,40.996,157.879
C07933=1045.812,336.311,382.992,172.724,40.992,157.878
C07934=1045.805,336.063,383.029,172.719,40.989,157.877
C07935=1045.798,335.816,383.064,172.715,40.985,157.876
C07936=1045.791,335.568,383.100,172.710,40.982,157.875
C07937=1045.784,335.321,383.136,172.706,40.978,157.874
C07938=1045.776,335.074,383.173,172.701,40.975,157.873
C07939=1045.770,334.826,383.208,172.697,40.971,157.872
C07940=1045.762,334.579,383.244,172.692,40.968,157.871
C07941=1045.755,334.332,383.279,172.687,40.965,157.870
C07942=1045.747,334.084,383.315,172.683,40.961,157.869
C07943=1045.738,333.768,383.361,172.678,40.957,157.868
C07944=1045.729,333.450,383.407,172.671,40.952,157.866
C07945=1045.721,333.134,383.453,172.666,40.948,157.865
C07946=1045.711,332.816,383.498,172.660,40.943,157.864
C07947=1045.703,332.569,383.534,172.655,40.940,157.863
C07948=1045.697,332.322,383.569,172.651,40.937,157.862
C07949=1045.690,332.075,383.605,172.647,40.933,157.861
C07950=1045.682,331.827,383.640,172.642,40.930,157.860
C07951=1045.675,331.579,383.675,172.638,40.926,157.859
C07952=1045.668,331.332,383.712,172.634,40.923,157.858
C07953=1045.661,331.085,383.747,172.629,40.919,157.857
C07954=1045.654,330.837,383.782,172.624,40.916,157.856
C07955=1045.647,330.590,383.818,172.620,40.913,157.855
C07956=1045.640,330.342,383.853,172.616,40.909,157.854
C07957=1045.633,330.095,383.888,172.611,40.906,157.853
C07958=1045.626,329.848,383.924,172.607,40.902,157.852
C07959=1045.619,329.601,383.959,172.603,40.899,157.851
C07960=1045.612,329.353,383.995,172.599,40.896,157.850
C07961=1045.605,329.105,384.030,172.594,40.893,157.849
C07962=1045.598,328.858,384.065,172.590,40.889,157.848
C07963=1045.590,328.610,384.100,172.586,40.886,157.847
C07964=1045.583,328.363,384.135,172.581,40.883,157.846
C07965=1045.577,328.116,384.170,172.577,40.880,157.845
C07966=1045.569,327.868,384.205,172.573,40.876,157.844
C07967=1045.562,327.620,384.240,172.569,40.873,157.843
C07968=1045.554,327.373,384.275,172.563,40.870,157.842
C07969=1045.548,327.126,384.310,172.559,40.866,157.841
C07970=1045.540,326.878,384.346,172.555,40.863,157.840
C07971=1045.533,326.631,384.380,172.551,40.860,157.839
C07972=1045.526,326.384,384.415,172.546,40.857,157.838
C07973=1045.518,326.137,384.450,172.542,40.854,157.837
C07974=1045.512,325.889,384.484,172.538,40.851,157.836
C07975=1045.505,325.640,384.520,172.534,40.847,157.835
C07976=1045.497,325.393,384.554,172.529,40.844,157.834
C07977=1045.490,325.146,384.589,172.525,40.841,157.833
C07978=1045.483,324.899,384.624,172.521,40.838,157.833
C07979=1045.476,324.652,384.659,172.517,40.835,157.832
C07980=1045.470,324.404,384.693,172.513,40.832,157.831
C07981=1045.461,324.156,384.728,172.508,40.828,157.830
C07982=1045.455,323.909,384.763,172.504,40.825,157.829
C07983=1045.447,323.661,384.798,172.500,40.822,157.828
C07984=1045.441,323.413,384.832,172.496,40.819,157.827
C07985=1045.434,323.166,384.868,172.492,40.816,157.826
C07986=1045.426,322.919,384.902,172.487,40.813,157.825
C07987=1045.420,322.671,384.937,172.483,40.809,157.824
C07988=1045.412,322.424,384.971,172.479,40.806,157.823
C07989=1045.406,322.176,385.005,172.475,40.803,157.822
C07990=1045.398,321.929,385.040,172.471,40.800,157.821
C07991=1045.392,321.682,385.075,172.467,40.797,157.820
C07992=1045.385,321.434,385.109,172.463,40.793,157.819
C07993=1045.378,321.187,385.144,172.458,40.791,157.819
C07994=1045.371,320.939,385.179,172.454,40.788,157.818
C07995=1045.364,320.692,385.213,172.450,40.784,157.817
C07996=1045.357,320.444,385.248,172.446,40.781,157.816
C07997=1045.350,320.197,385.282,172.442,40.778,157.815
C07998=1045.343,319.949,385.316,172.438,40.775,157.814
C07999=1045.334,319.627,385.361,172.433,40.771,157.813
C08000=1045.325,319.305,385.406,172.427,40.767,157.812
C08001=1045.316,318.982,385.451,172.422,40.763,157.810
C08002=1045.307,318.661,385.495,172.417,40.759,157.809
C08003=1045.300,318.413,385.530,172.413,40.756,157.808
C08004=1045.293,318.166,385.564,172.409,40.752,157.807
C08005=1045.286,317.918,385.599,172.405,40.749,157.807
C08006=1045.280,317.671,385.632,172.401,40.747,157.806
C08007=1045.273,317.423,385.667,172.396,40.744,157.805
C08008=1045.266,317.176,385.701,172.392,40.740,157.804
C08009=1045.259,316.928,385.735,172.388,40.737,157.803
C08010=1045.253,316.680,385.771,172.384,40.734,157.802
C08011=1045.245,316.433,385.804,172.380,40.731,157.801
C08012=1045.239,316.186,385.838,172.376,40.728,157.800
C08013=1045.232,315.938,385.872,172.372,40.725,157.799
C08014=1045.225,315.690,385.906,172.368,40.722,157.799
C08015=1045.218,315.443,385.941,172.364,40.719,157.798
C08016=1045.212,315.196,385.975,172.360,40.716,157.797
C08017=1045.205,314.948,386.009,172.356,40.713,157.796
C08018=1045.198,314.700,386.043,172.352,40.710,157.795
C08019=1045.192,314.452,386.077,172.348,40.707,157.794
C08020=1045.185,314.205,386.111,172.344,40.704,157.793
C08021=1045.179,313.957,386.145,172.340,40.701,157.792
C08022=1045.171,313.709,386.179,172.336,40.698,157.792
C08023=1045.166,313.462,386.213,172.333,40.695,157.791
C08024=1045.158,313.215,386.248,172.329,40.692,157.790
C08025=1045.152,312.967,386.282,172.325,40.688,157.789
C08026=1045.145,312.720,386.316,172.321,40.686,157.788
C08027=1045.138,312.472,386.349,172.317,40.683,157.787
C08028=1045.131,312.224,386.382,172.313,40.680,157.786
C08029=1045.124,311.976,386.416,172.309,40.677,157.786
C08030=1045.117,311.729,386.450,172.305,40.674,157.785
C08031=1045.110,311.482,386.484,172.301,40.671,157.784
C08032=1045.103,311.234,386.517,172.297,40.668,157.783
C08033=1045.096,310.986,386.550,172.293,40.666,157.782
C08034=1045.089,310.739,386.584,172.290,40.663,157.782
C08035=1045.082,310.491,386.618,172.286,40.660,157.781
C08036=1045.075,310.243,386.651,172.282,40.657,157.780
C08037=1045.068,309.995,386.685,172.278,40.654,157.779
C08038=1045.061,309.749,386.718,172.275,40.651,157.778
C08039=1045.054,309.500,386.751,172.271,40.648,157.777
C08040=1045.046,309.253,386.785,172.267,40.646,157.777
C08041=1045.040,309.006,386.818,172.263,40.643,157.776
C08042=1045.033,308.757,386.851,172.259,40.640,157.775
C08043=1045.026,308.510,386.885,172.256,40.637,157.774
C08044=1045.020,308.262,386.918,172.252,40.634,157.773
C08045=1045.012,308.014,386.951,172.248,40.631,157.772
C08046=1045.006,307.767,386.985,172.244,40.629,157.772
C08047=1044.998,307.519,387.017,172.240,40.626,157.771
C08048=1044.991,307.272,387.051,172.236,40.623,157.770
C08049=1044.985,307.024,387.084,172.232,40.620,157.769
C08050=1044.977,306.776,387.118,172.228,40.618,157.768
C08051=1044.971,306.529,387.151,172.225,40.615,157.768
C08052=1044.964,306.281,387.184,172.221,40.612,157.767
C08053=1044.958,306.034,387.217,172.218,40.609,157.766
C08054=1044.950,305.786,387.250,172.214,40.606,157.765
C08055=1044.941,305.468,387.292,172.209,40.603,157.764
C08056=1044.933,305.151,387.335,172.204,40.599,157.763
C08057=1044.924,304.834,387.377,172.200,40.596,157.762
C08058=1044.915,304.516,387.420,172.194,40.592,157.761
C08059=1044.908,304.269,387.453,172.191,40.589,157.760
C08060=1044.901,304.021,387.486,172.187,40.587,157.760
C08061=1044.895,303.773,387.519,172.183,40.584,157.759
C08062=1044.889,303.526,387.552,172.179,40.581,157.758
C08063=1044.882,303.277,387.585,172.176,40.578,157.757
C08064=1044.874,303.031,387.618,172.172,40.575,157.756
C08065=1044.868,302.783,387.651,172.169,40.573,157.756
C08066=1044.861,302.535,387.684,172.165,40.570,157.755
C08067=1044.854,302.287,387.717,172.161,40.567,157.754
C08068=1044.848,302.040,387.750,172.157,40.565,157.753
C08069=1044.841,301.792,387.783,172.154,40.561,157.752
C08070=1044.834,301.544,387.816,172.150,40.559,157.752
C08071=1044.828,301.296,387.848,172.146,40.556,157.751
C08072=1044.821,301.048,387.881,172.143,40.553,157.750
C08073=1044.814,300.801,387.914,172.139,40.551,157.749
C08074=1044.808,300.554,387.948,172.136,40.548,157.748
C08075=1044.801,300.305,387.981,172.132,40.545,157.748
C08076=1044.794,300.058,388.013,172.128,40.543,157.747
C08077=1044.788,299.810,388.046,172.125,40.540,157.746
C08078=1044.781,299.563,388.078,172.122,40.536,157.745
C08079=1044.774,299.315,388.111,172.118,40.534,157.745
C08080=1044.768,299.067,388.144,172.114,40.531,157.744
C08081=1044.761,298.820,388.176,172.110,40.528,157.743
C08082=1044.754,298.571,388.209,172.107,40.526,157.742
C08083=1044.748,298.324,388.242,172.104,40.523,157.741
C08084=1044.742,298.076,388.275,172.100,40.520,157.741
C08085=1044.735,297.829,388.307,172.096,40.518,157.740
C08086=1044.728,297.581,388.340,172.093,40.515,157.739
C08087=1044.721,297.333,388.373,172.089,40.512,157.738
C08088=1044.715,297.085,388.406,172.085,40.510,157.738
C08089=1044.709,296.838,388.438,172.082,40.507,157.737
C08090=1044.701,296.589,388.470,172.079,40.504,157.736
C08091=1044.695,296.342,388.503,172.075,40.501,157.735
C08092=1044.689,296.094,388.536,172.071,40.499,157.735
C08093=1044.683,295.846,388.568,172.068,40.496,157.734
C08094=1044.676,295.599,388.601,172.065,40.493,157.733
C08095=1044.669,295.350,388.633,172.061,40.491,157.732
C08096=1044.662,295.103,388.665,172.057,40.488,157.732
C08097=1044.656,294.855,388.698,172.054,40.485,157.731
C08098=1044.649,294.608,388.730,172.050,40.483,157.730
C08099=1044.642,294.359,388.762,172.046,40.480,157.729
C08100=1044.635,294.112,388.795,172.044,40.477,157.729
C08101=1044.629,293.864,388.827,172.040,40.475,157.728
C08102=1044.622,293.616,388.859,172.036,40.472,157.727
C08103=1044.615,293.369,388.891,172.032,40.470,157.726
C08104=1044.608,293.120,388.923,172.030,40.467,157.726
C08105=1044.601,292.873,388.955,172.026,40.464,157.725
C08106=1044.595,292.625,388.987,172.022,40.462,157.724
C08107=1044.588,292.377,389.020,172.019,40.459,157.723
C08108=1044.582,292.130,389.051,172.016,40.457,157.723
C08109=1044.575,291.882,389.083,172.012,40.454,157.722
C08110=1044.568,291.633,389.116,172.009,40.452,157.721
C08111=1044.560,291.333,389.155,172.004,40.449,157.720
C08112=1044.551,291.031,389.193,172.000,40.445,157.720
C08113=1044.543,290.731,389.232,171.996,40.442,157.719
C08114=1044.535,290.430,389.271,171.992,40.439,157.718
C08115=1044.529,290.182,389.303,171.989,40.437,157.717
C08116=1044.522,289.934,389.335,171.985,40.434,157.716
C08117=1044.515,289.686,389.367,171.982,40.431,157.716
C08118=1044.509,289.438,389.399,171.978,40.429,157.715
C08119=1044.502,289.190,389.431,171.975,40.426,157.714
C08120=1044.495,288.943,389.462,171.972,40.424,157.713
C08121=1044.488,288.695,389.494,171.968,40.421,157.713
C08122=1044.482,288.447,389.526,171.965,40.419,157.712
C08123=1044.475,288.199,389.558,171.961,40.416,157.711
C08124=1044.469,287.951,389.589,171.958,40.413,157.711
C08125=1044.462,287.703,389.621,171.955,40.411,157.710
C08126=1044.456,287.456,389.653,171.951,40.409,157.709
C08127=1044.449,287.208,389.685,171.948,40.406,157.708
C08128=1044.442,286.960,389.716,171.945,40.404,157.708
C08129=1044.435,286.711,389.748,171.941,40.401,157.707
C08130=1044.428,286.463,389.780,171.938,40.398,157.706
C08131=1044.421,286.215,389.811,171.934,40.396,157.706
C08132=1044.414,285.968,389.843,171.932,40.393,157.705
C08133=1044.408,285.720,389.875,171.928,40.391,157.704
C08134=1044.401,285.472,389.906,171.924,40.389,157.704
C08135=1044.394,285.225,389.937,171.922,40.386,157.703
C08136=1044.387,284.977,389.969,171.918,40.384,157.702
C08137=1044.381,284.729,390.000,171.915,40.381,157.701
C08138=1044.374,284.481,390.032,171.911,40.379,157.701
C08139=1044.367,284.233,390.063,171.908,40.376,157.700
C08140=1044.361,283.985,390.095,171.905,40.374,157.699
C08141=1044.354,283.737,390.126,171.901,40.371,157.699
C08142=1044.347,283.489,390.157,171.899,40.369,157.698
C08143=1044.340,283.241,390.189,171.895,40.366,157.697
C08144=1044.334,282.993,390.220,171.892,40.364,157.697
C08145=1044.327,282.745,390.252,171.888,40.361,157.696
C08146=1044.320,282.497,390.282,171.885,40.359,157.695
C08147=1044.314,282.250,390.314,171.882,40.356,157.695
C08148=1044.308,282.002,390.345,171.879,40.354,157.694
C08149=1044.301,281.754,390.376,171.875,40.352,157.693
C08150=1044.294,281.506,390.408,171.872,40.349,157.693
C08151=1044.287,281.258,390.439,171.869,40.347,157.692
C08152=1044.281,281.010,390.471,171.865,40.344,157.691
C08153=1044.274,280.762,390.501,171.863,40.342,157.691
C08154=1044.268,280.514,390.533,171.859,40.339,157.690
C08155=1044.261,280.266,390.564,171.856,40.337,157.689
C08156=1044.255,280.019,390.595,171.852,40.334,157.688
C08157=1044.248,279.771,390.627,171.850,40.332,157.688
C08158=1044.242,279.522,390.658,171.846,40.329,157.687
C08159=1044.235,279.274,390.689,171.843,40.327,157.687
C08160=1044.228,279.026,390.720,171.840,40.324,157.686
C08161=1044.222,278.778,390.751,171.837,40.322,157.685
C08162=1044.215,278.530,390.783,171.834,40.319,157.684
C08163=1044.209,278.283,390.814,171.830,40.317,157.684
C08164=1044.202,278.034,390.844,171.828,40.314,157.683
C08165=1044.195,277.787,390.875,171.824,40.312,157.682
C08166=1044.188,277.539,390.907,171.821,40.310,157.682
C08167=1044.181,277.249,390.942,171.817,40.307,157.681
C08168=1044.173,276.960,390.979,171.814,40.304,157.680
C08169=1044.165,276.670,391.014,171.810,40.301,157.679
C08170=1044.157,276.381,391.050,171.806,40.299,157.679
C08171=1044.151,276.133,391.081,171.803,40.296,157.678
C08172=1044.144,275.885,391.112,171.800,40.294,157.677
C08173=1044.138,275.636,391.143,171.797,40.292,157.677
C08174=1044.130,275.389,391.174,171.793,40.289,157.676
C08175=1044.124,275.141,391.204,171.791,40.287,157.675
C08176=1044.118,274.893,391.236,171.787,40.285,157.675
C08177=1044.111,274.645,391.266,171.784,40.282,157.674
C08178=1044.104,274.397,391.297,171.782,40.280,157.673
C08179=1044.098,274.149,391.328,171.778,40.277,157.673
C08180=1044.092,273.901,391.358,171.775,40.275,157.672
C08181=1044.084,273.653,391.389,171.771,40.272,157.671
C08182=1044.078,273.405,391.420,171.769,40.270,157.671
C08183=1044.072,273.157,391.451,171.765,40.268,157.670
C08184=1044.064,272.909,391.481,171.762,40.265,157.670
C08185=1044.058,272.661,391.512,171.760,40.263,157.669
C08186=1044.051,272.413,391.543,171.756,40.260,157.668
C08187=1044.045,272.165,391.573,171.753,40.258,157.668
C08188=1044.038,271.917,391.604,171.750,40.256,157.667
C08189=1044.032,271.668,391.634,171.747,40.253,157.666
C08190=1044.025,271.421,391.665,171.744,40.251,157.666
C08191=1044.019,271.173,391.696,171.741,40.249,157.665
C08192=1044.012,270.925,391.726,171.738,40.247,157.664
C08193=1044.006,270.677,391.756,171.735,40.244,157.664
C08194=1043.999,270.429,391.786,171.732,40.242,157.663
C08195=1043.992,270.180,391.817,171.729,40.240,157.662
C08196=1043.985,269.932,391.848,171.725,40.237,157.662
C08197=1043.979,269.685,391.878,171.723,40.235,157.661
C08198=1043.972,269.436,391.908,171.720,40.232,157.661
C08199=1043.965,269.188,391.939,171.716,40.230,157.660
C08200=1043.959,268.940,391.969,171.714,40.227,157.659
C08201=1043.952,268.692,391.999,171.711,40.225,157.659
C08202=1043.946,268.444,392.029,171.707,40.223,157.658
C08203=1043.939,268.196,392.060,171.705,40.221,157.657
C08204=1043.932,267.948,392.090,171.702,40.219,157.657
C08205=1043.926,267.700,392.120,171.698,40.216,157.656
C08206=1043.919,267.452,392.150,171.696,40.214,157.655
C08207=1043.912,267.203,392.181,171.692,40.212,157.655
C08208=1043.906,266.955,392.211,171.689,40.209,157.654
C08209=1043.899,266.707,392.241,171.687,40.207,157.654
C08210=1043.892,266.460,392.271,171.683,40.204,157.653
C08211=1043.886,266.211,392.302,171.680,40.202,157.652
C08212=1043.879,265.963,392.332,171.678,40.200,157.652
C08213=1043.872,265.716,392.361,171.675,40.198,157.651
C08214=1043.866,265.467,392.392,171.672,40.196,157.651
C08215=1043.859,265.219,392.422,171.669,40.193,157.650
C08216=1043.853,264.971,392.451,171.666,40.191,157.649
C08217=1043.847,264.723,392.482,171.663,40.188,157.649
C08218=1043.840,264.475,392.512,171.660,40.186,157.648
C08219=1043.832,264.226,392.542,171.657,40.184,157.647
C08220=1043.827,263.979,392.572,171.654,40.182,157.647
C08221=1043.819,263.730,392.602,171.651,40.179,157.646
C08222=1043.813,263.482,392.631,171.648,40.177,157.645
C08223=1043.805,263.198,392.667,171.645,40.174,157.645
C08224=1043.798,262.913,392.701,171.642,40.172,157.644
C08225=1043.791,262.628,392.735,171.638,40.169,157.643
C08226=1043.783,262.342,392.770,171.634,40.166,157.643
C08227=1043.777,262.095,392.800,171.632,40.164,157.642
C08228=1043.770,261.846,392.829,171.629,40.162,157.641
C08229=1043.763,261.598,392.859,171.627,40.160,157.641
C08230=1043.756,261.350,392.888,171.623,40.158,157.640
C08231=1043.749,261.102,392.918,171.620,40.155,157.640
C08232=1043.743,260.854,392.948,171.618,40.153,157.639
C08233=1043.736,260.605,392.977,171.614,40.151,157.638
C08234=1043.729,260.358,393.007,171.611,40.149,157.638
C08235=1043.722,260.109,393.037,171.609,40.147,157.637
C08236=1043.716,259.861,393.066,171.606,40.144,157.637
C08237=1043.709,259.612,393.096,171.603,40.142,157.636
C08238=1043.702,259.365,393.125,171.600,40.140,157.635
C08239=1043.696,259.116,393.155,171.597,40.138,157.635
C08240=1043.688,258.869,393.184,171.595,40.135,157.634
C08241=1043.681,258.620,393.213,171.591,40.133,157.634
C08242=1043.675,258.373,393.243,171.589,40.131,157.633
C08243=1043.668,258.124,393.273,171.586,40.129,157.633
C08244=1043.662,257.876,393.302,171.583,40.127,157.632
C08245=1043.655,257.627,393.332,171.580,40.125,157.631
C08246=1043.648,257.379,393.361,171.577,40.122,157.631
C08247=1043.641,257.131,393.391,171.574,40.120,157.630
C08248=1043.635,256.883,393.420,171.572,40.118,157.630
C08249=1043.628,256.634,393.449,171.568,40.116,157.629
C08250=1043.622,256.387,393.479,171.566,40.113,157.628
C08251=1043.615,256.138,393.508,171.563,40.111,157.628
C08252=1043.608,255.890,393.538,171.560,40.109,157.627
C08253=1043.602,255.642,393.567,171.558,40.107,157.627
C08254=1043.595,255.393,393.597,171.554,40.105,157.626
C08255=1043.588,255.145,393.625,171.552,40.102,157.625
C08256=1043.581,254.898,393.655,171.549,40.100,157.625
C08257=1043.575,254.649,393.684,171.546,40.098,157.624
C08258=1043.568,254.401,393.713,171.544,40.096,157.624
C08259=1043.562,254.153,393.742,171.540,40.094,157.623
C08260=1043.555,253.905,393.773,171.538,40.091,157.622
C08261=1043.549,253.657,393.802,171.535,40.089,157.622
C08262=1043.542,253.408,393.831,171.532,40.087,157.621
C08263=1043.536,253.160,393.860,171.530,40.085,157.621
C08264=1043.529,252.912,393.890,171.527,40.082,157.620
C08265=1043.523,252.664,393.919,171.524,40.079,157.619
C08266=1043.515,252.415,393.948,171.521,40.077,157.619
C08267=1043.509,252.167,393.977,171.518,40.075,157.618
C08268=1043.503,251.919,394.006,171.515,40.073,157.618
C08269=1043.496,251.670,394.035,171.513,40.071,157.617
C08270=1043.490,251.422,394.064,171.510,40.068,157.616
C08271=1043.483,251.175,394.094,171.508,40.066,157.616
C08272=1043.476,250.926,394.123,171.505,40.064,157.615
C08273=1043.470,250.678,394.152,171.501,40.062,157.615
C08274=1043.464,250.430,394.181,171.499,40.059,157.614
C08275=1043.457,250.182,394.210,171.496,40.057,157.613
C08276=1043.450,249.933,394.239,171.494,40.055,157.613
C08277=1043.444,249.685,394.268,171.491,40.053,157.612
C08278=1043.437,249.437,394.297,171.488,40.050,157.612
C08279=1043.430,249.150,394.331,171.486,40.048,157.611
C08280=1043.423,248.864,394.364,171.482,40.045,157.610
C08281=1043.415,248.577,394.398,171.479,40.043,157.610
C08282=1043.408,248.291,394.431,171.476,40.040,157.609
C08283=1043.401,248.042,394.460,171.473,40.038,157.608
C08284=1043.394,247.794,394.489,171.470,40.036,157.608
C08285=1043.388,247.546,394.518,171.468,40.033,157.607
C08286=1043.382,247.298,394.547,171.465,40.031,157.607
C08287=1043.376,247.050,394.576,171.463,40.029,157.606
C08288=1043.370,246.802,394.605,171.460,40.026,157.605
C08289=1043.362,246.553,394.634,171.457,40.024,157.605
C08290=1043.356,246.305,394.663,171.455,40.022,157.604
C08291=1043.349,246.057,394.692,171.452,40.020,157.604
C08292=1043.343,245.809,394.721,171.450,40.017,157.603
C08293=1043.337,245.561,394.750,171.447,40.015,157.602
C08294=1043.331,245.312,394.779,171.444,40.013,157.602
C08295=1043.323,245.063,394.808,171.442,40.011,157.601
C08296=1043.317,244.815,394.837,171.439,40.008,157.601
C08297=1043.310,244.568,394.865,171.437,40.006,157.600
C08298=1043.304,244.319,394.893,171.434,40.004,157.600
C08299=1043.298,244.071,394.922,171.430,40.002,157.599
C08300=1043.291,243.823,394.951,171.428,39.999,157.598
C08301=1043.285,243.575,394.980,171.425,39.998,157.598
C08302=1043.277,243.326,395.008,171.423,39.996,157.597
C08303=1043.271,243.077,395.037,171.420,39.993,157.597
C08304=1043.265,242.829,395.066,171.417,39.991,157.596
C08305=1043.258,242.581,395.094,171.415,39.989,157.596
C08306=1043.252,242.333,395.123,171.412,39.987,157.595
C08307=1043.245,242.085,395.151,171.410,39.984,157.594
C08308=1043.239,241.836,395.180,171.407,39.982,157.594
C08309=1043.233,241.588,395.209,171.404,39.980,157.593
C08310=1043.226,241.340,395.237,171.402,39.978,157.593
C08311=1043.219,241.091,395.266,171.399,39.975,157.592
C08312=1043.212,240.843,395.294,171.397,39.973,157.592
C08313=1043.206,240.594,395.322,171.394,39.971,157.591
C08314=1043.199,240.346,395.351,171.391,39.969,157.590
C08315=1043.193,240.098,395.379,171.389,39.967,157.590
C08316=1043.186,239.850,395.407,171.386,39.965,157.589
C08317=1043.180,239.601,395.436,171.384,39.962,157.589
C08318=1043.173,239.354,395.464,171.381,39.960,157.588
C08319=1043.167,239.105,395.492,171.379,39.958,157.588
C08320=1043.159,238.856,395.521,171.376,39.956,157.587
C08321=1043.153,238.608,395.549,171.373,39.953,157.586
C08322=1043.146,238.360,395.578,171.371,39.952,157.586
C08323=1043.140,238.111,395.606,171.368,39.949,157.585
C08324=1043.133,237.863,395.633,171.366,39.947,157.585
C08325=1043.127,237.615,395.662,171.363,39.945,157.584
C08326=1043.120,237.366,395.690,171.361,39.943,157.584
C08327=1043.113,237.118,395.718,171.358,39.940,157.583
C08328=1043.106,236.870,395.746,171.355,39.938,157.582
C08329=1043.100,236.621,395.775,171.354,39.936,157.582
C08330=1043.094,236.373,395.802,171.351,39.934,157.581
C08331=1043.087,236.125,395.831,171.349,39.932,157.581
C08332=1043.080,235.876,395.859,171.346,39.930,157.580
C08333=1043.074,235.628,395.887,171.344,39.927,157.580
C08334=1043.067,235.380,395.915,171.341,39.925,157.579
C08335=1043.059,235.087,395.948,171.338,39.923,157.579
C08336=1043.051,234.795,395.981,171.335,39.920,157.578
C08337=1043.044,234.503,396.015,171.332,39.918,157.577
C08338=1043.036,234.211,396.047,171.329,39.915,157.577
C08339=1043.029,233.963,396.076,171.327,39.913,157.576
C08340=1043.023,233.714,396.103,171.324,39.910,157.575
C08341=1043.017,233.466,396.132,171.322,39.908,157.575
C08342=1043.010,233.217,396.159,171.319,39.906,157.574
C08343=1043.004,232.969,396.187,171.317,39.904,157.574
C08344=1042.997,232.721,396.216,171.314,39.902,157.573
C08345=1042.991,232.472,396.244,171.311,39.900,157.573
C08346=1042.984,232.224,396.272,171.309,39.897,157.572
C08347=1042.977,231.975,396.299,171.307,39.895,157.571
C08348=1042.971,231.727,396.327,171.305,39.893,157.571
C08349=1042.964,231.479,396.354,171.302,39.891,157.570
C08350=1042.958,231.231,396.382,171.300,39.889,157.570
C08351=1042.952,230.982,396.410,171.297,39.887,157.569
C08352=1042.945,230.734,396.439,171.294,39.884,157.569
C08353=1042.938,230.486,396.467,171.292,39.882,157.568
C08354=1042.931,230.237,396.494,171.289,39.880,157.568
C08355=1042.925,229.989,396.522,171.288,39.877,157.567
C08356=1042.918,229.740,396.550,171.285,39.875,157.566
C08357=1042.911,229.492,396.578,171.283,39.874,157.566
C08358=1042.905,229.243,396.605,171.280,39.871,157.565
C08359=1042.898,228.995,396.633,171.277,39.869,157.565
C08360=1042.892,228.747,396.660,171.275,39.867,157.564
C08361=1042.886,228.498,396.689,171.272,39.864,157.564
C08362=1042.879,228.250,396.716,171.270,39.862,157.563
C08363=1042.872,228.001,396.743,171.268,39.860,157.563
C08364=1042.866,227.753,396.771,171.266,39.858,157.562
C08365=1042.859,227.504,396.798,171.263,39.856,157.562
C08366=1042.852,227.256,396.826,171.260,39.854,157.561
C08367=1042.846,227.007,396.854,171.258,39.852,157.561
C08368=1042.839,226.759,396.882,171.255,39.850,157.560
C08369=1042.833,226.511,396.909,171.253,39.847,157.559
C08370=1042.826,226.262,396.936,171.251,39.845,157.559
C08371=1042.819,226.014,396.963,171.249,39.843,157.558
C08372=1042.812,225.766,396.991,171.246,39.841,157.558
C08373=1042.806,225.517,397.018,171.244,39.839,157.557
C08374=1042.799,225.269,397.046,171.241,39.837,157.557
C08375=1042.792,225.020,397.074,171.238,39.834,157.556
C08376=1042.786,224.772,397.101,171.237,39.832,157.555
C08377=1042.780,224.524,397.128,171.234,39.830,157.555
C08378=1042.772,224.275,397.155,171.232,39.828,157.554
C08379=1042.766,224.027,397.183,171.229,39.826,157.554
C08380=1042.759,223.778,397.210,171.227,39.823,157.553
C08381=1042.753,223.530,397.238,171.225,39.821,157.553
C08382=1042.747,223.282,397.265,171.223,39.819,157.552
C08383=1042.740,223.033,397.292,171.220,39.817,157.552
C08384=1042.734,222.784,397.320,171.218,39.815,157.551
C08385=1042.727,222.536,397.348,171.215,39.813,157.551
C08386=1042.720,222.288,397.375,171.213,39.810,157.550
C08387=1042.714,222.039,397.402,171.211,39.808,157.549
C08388=1042.707,221.791,397.429,171.208,39.806,157.549
C08389=1042.701,221.542,397.456,171.206,39.804,157.548
C08390=1042.694,221.294,397.484,171.204,39.802,157.548
C08391=1042.686,220.995,397.516,171.201,39.799,157.547
C08392=1042.678,220.695,397.549,171.198,39.796,157.546
C08393=1042.671,220.395,397.582,171.195,39.794,157.546
C08394=1042.662,220.095,397.615,171.192,39.791,157.545
C08395=1042.656,219.847,397.642,171.190,39.789,157.545
C08396=1042.649,219.599,397.669,171.188,39.787,157.544
C08397=1042.643,219.350,397.696,171.186,39.784,157.544
C08398=1042.636,219.101,397.724,171.183,39.782,157.543
C08399=1042.629,218.853,397.750,171.181,39.780,157.542
C08400=1042.623,218.605,397.778,171.179,39.778,157.542
C08401=1042.616,218.356,397.804,171.177,39.776,157.541
C08402=1042.609,218.108,397.832,171.174,39.774,157.541
C08403=1042.602,217.859,397.858,171.172,39.771,157.540
C08404=1042.596,217.610,397.885,171.170,39.770,157.540
C08405=1042.589,217.362,397.913,171.168,39.767,157.539
C08406=1042.583,217.114,397.939,171.165,39.765,157.539
C08407=1042.576,216.865,397.967,171.162,39.763,157.538
C08408=1042.569,216.617,397.993,171.161,39.760,157.538
C08409=1042.562,216.368,398.021,171.158,39.759,157.537
C08410=1042.557,216.120,398.047,171.156,39.756,157.537
C08411=1042.549,215.871,398.074,171.154,39.754,157.536
C08412=1042.543,215.623,398.101,171.152,39.752,157.535
C08413=1042.536,215.375,398.128,171.149,39.749,157.535
C08414=1042.530,215.126,398.155,171.147,39.748,157.534
C08415=1042.522,214.878,398.182,171.145,39.745,157.534
C08416=1042.517,214.629,398.208,171.143,39.743,157.533
C08417=1042.510,214.380,398.235,171.140,39.741,157.533
C08418=1042.503,214.133,398.262,171.138,39.738,157.532
C08419=1042.497,213.884,398.289,171.136,39.736,157.532
C08420=1042.490,213.635,398.316,171.133,39.735,157.531
C08421=1042.484,213.386,398.342,171.132,39.732,157.531
C08422=1042.477,213.138,398.369,171.129,39.730,157.530
C08423=1042.470,212.889,398.396,171.127,39.728,157.529
C08424=1042.464,212.641,398.422,171.125,39.725,157.529
C08425=1042.458,212.392,398.449,171.123,39.723,157.528
C08426=1042.451,212.145,398.476,171.120,39.721,157.528
C08427=1042.444,211.896,398.503,171.119,39.719,157.527
C08428=1042.438,211.648,398.529,171.116,39.717,157.527
C08429=1042.431,211.399,398.556,171.113,39.714,157.526
C08430=1042.424,211.150,398.583,171.112,39.712,157.526
C08431=1042.418,210.902,398.610,171.109,39.710,157.525
C08432=1042.411,210.653,398.636,171.107,39.708,157.525
C08433=1042.405,210.405,398.663,171.105,39.706,157.524
C08434=1042.398,210.156,398.690,171.103,39.703,157.524
C08435=1042.391,209.907,398.716,171.100,39.701,157.523
C08436=1042.385,209.659,398.743,171.099,39.699,157.522
C08437=1042.378,209.410,398.769,171.096,39.697,157.522
C08438=1042.372,209.162,398.795,171.094,39.695,157.521
C08439=1042.365,208.913,398.822,171.092,39.692,157.521
C08440=1042.359,208.665,398.848,171.089,39.690,157.520
C08441=1042.352,208.416,398.875,171.088,39.688,157.520
C08442=1042.345,208.168,398.901,171.085,39.686,157.519
C08443=1042.339,207.919,398.928,171.083,39.684,157.519
C08444=1042.332,207.671,398.954,171.081,39.681,157.518
C08445=1042.325,207.423,398.980,171.079,39.679,157.518
C08446=1042.319,207.173,399.007,171.076,39.677,157.517
C08447=1042.311,206.880,399.038,171.075,39.674,157.516
C08448=1042.303,206.586,399.070,171.072,39.672,157.516
C08449=1042.295,206.292,399.100,171.069,39.669,157.515
C08450=1042.287,205.997,399.132,171.067,39.667,157.515
C08451=1042.259,204.859,399.247,170.790,39.564,157.484
C08452=1042.253,204.632,399.270,170.787,39.563,157.483
C08453=1042.247,204.405,399.293,170.785,39.561,157.483
C08454=1042.242,204.177,399.316,170.782,39.560,157.483
C08455=1042.236,203.928,399.341,170.779,39.558,157.482
C08456=1042.230,203.679,399.366,170.777,39.556,157.482
C08457=1042.224,203.431,399.392,170.773,39.555,157.481
C08458=1042.218,203.183,399.417,170.771,39.554,157.481
C08459=1042.211,202.935,399.441,170.767,39.552,157.480
C08460=1042.205,202.685,399.466,170.764,39.551,157.480
C08461=1042.199,202.437,399.491,170.762,39.549,157.480
C08462=1042.193,202.188,399.517,170.758,39.548,157.479
C08463=1042.186,201.939,399.542,170.756,39.547,157.479
C08464=1042.181,201.691,399.566,170.753,39.545,157.479
C08465=1042.175,201.442,399.592,170.750,39.544,157.478
C08466=1042.169,201.193,399.617,170.747,39.542,157.478
C08467=1042.162,200.944,399.641,170.744,39.541,157.477
C08468=1042.156,200.696,399.666,170.741,39.540,157.477
C08469=1042.150,200.447,399.692,170.739,39.539,157.477
C08470=1042.144,200.199,399.715,170.735,39.537,157.476
C08471=1042.137,199.950,399.741,170.733,39.536,157.476
C08472=1042.131,199.701,399.765,170.730,39.534,157.476
C08473=1042.125,199.452,399.790,170.727,39.533,157.475
C08474=1042.118,199.204,399.815,170.724,39.532,157.475
C08475=1042.112,198.955,399.839,170.722,39.531,157.475
C08476=1042.106,198.707,399.864,170.718,39.529,157.474
C08477=1042.100,198.458,399.888,170.715,39.528,157.474
C08478=1042.093,198.209,399.914,170.713,39.527,157.473
C08479=1042.087,197.960,399.938,170.709,39.525,157.473
C08480=1042.080,197.711,399.963,170.707,39.524,157.473
C08481=1042.075,197.463,399.987,170.704,39.523,157.472
C08482=1042.068,197.215,400.012,170.701,39.521,157.472
C08483=1042.062,196.965,400.037,170.698,39.520,157.472
C08484=1042.056,196.716,400.061,170.696,39.519,157.471
C08485=1042.050,196.468,400.086,170.692,39.518,157.471
C08486=1042.043,196.219,400.110,170.690,39.516,157.470
C08487=1042.037,195.971,400.135,170.687,39.515,157.470
C08488=1042.031,195.721,400.160,170.684,39.514,157.470
C08489=1042.025,195.473,400.183,170.682,39.512,157.469
C08490=1042.019,195.224,400.209,170.679,39.511,157.469
C08491=1042.012,194.975,400.233,170.676,39.510,157.469
C08492=1042.007,194.727,400.258,170.673,39.509,157.468
C08493=1042.000,194.478,400.282,170.671,39.508,157.468
C08494=1041.994,194.229,400.306,170.667,39.506,157.468
C08495=1041.987,193.924,400.337,170.664,39.505,157.467
C08496=1041.979,193.619,400.366,170.660,39.503,157.467
C08497=1041.972,193.314,400.396,170.657,39.502,157.466
C08498=1041.964,193.008,400.427,170.654,39.500,157.466
C08499=1041.958,192.761,400.451,170.651,39.499,157.466
C08500=1041.952,192.511,400.476,170.648,39.497,157.465
C08501=1041.946,192.262,400.500,170.646,39.496,157.465
C08502=1041.940,192.014,400.524,170.642,39.495,157.465
C08503=1041.933,191.765,400.549,170.640,39.493,157.464
C08504=1041.927,191.516,400.573,170.638,39.492,157.464
C08505=1041.921,191.268,400.597,170.634,39.491,157.464
C08506=1041.916,191.018,400.622,170.632,39.490,157.463
C08507=1041.909,190.770,400.645,170.629,39.489,157.463
C08508=1041.904,190.521,400.670,170.626,39.488,157.463
C08509=1041.897,190.273,400.695,170.624,39.486,157.462
C08510=1041.891,190.024,400.719,170.621,39.485,157.462
C08511=1041.884,189.739,400.746,170.617,39.483,157.461
C08512=1041.877,189.455,400.774,170.615,39.482,157.461
C08513=1041.870,189.171,400.801,170.612,39.481,157.461
C08514=1041.864,188.886,400.830,170.608,39.480,157.460
C08515=1041.857,188.637,400.854,170.606,39.478,157.460
C08516=1041.852,188.389,400.878,170.603,39.477,157.460
C08517=1041.845,188.140,400.902,170.600,39.476,157.459
C08518=1041.840,187.891,400.926,170.598,39.474,157.459
C08519=1041.833,187.642,400.950,170.595,39.473,157.459
C08520=1041.828,187.393,400.975,170.592,39.472,157.458
C08521=1041.821,187.144,400.999,170.590,39.471,157.458
C08522=1041.816,186.896,401.023,170.587,39.469,157.457
C08523=1041.809,186.647,401.047,170.584,39.468,157.457
C08524=1041.803,186.399,401.071,170.581,39.467,157.457
C08525=1041.798,186.149,401.095,170.579,39.465,157.456
C08526=1041.792,185.901,401.119,170.576,39.464,157.456
C08527=1041.786,185.652,401.144,170.573,39.463,157.456
C08528=1041.780,185.404,401.167,170.571,39.462,157.456
C08529=1041.774,185.155,401.192,170.568,39.461,157.455
C08530=1041.768,184.906,401.216,170.565,39.460,157.455
C08531=1041.762,184.657,401.240,170.563,39.458,157.455
C08532=1041.756,184.408,401.264,170.560,39.457,157.454
C08533=1041.750,184.160,401.288,170.557,39.456,157.454
C08534=1041.744,183.911,401.312,170.555,39.455,157.453
C08535=1041.738,183.662,401.336,170.552,39.454,157.453
C08536=1041.732,183.413,401.360,170.549,39.453,157.453
C08537=1041.726,183.164,401.383,170.547,39.451,157.453
C08538=1041.719,182.915,401.407,170.545,39.450,157.452
C08539=1041.713,182.667,401.431,170.541,39.449,157.452
C08540=1041.706,182.418,401.454,170.539,39.448,157.452
C08541=1041.700,182.170,401.477,170.536,39.447,157.451
C08542=1041.694,181.921,401.501,170.534,39.446,157.451
C08543=1041.688,181.672,401.524,170.531,39.445,157.451
C08544=1041.681,181.423,401.548,170.528,39.444,157.450
C08545=1041.675,181.174,401.572,170.526,39.443,157.450
C08546=1041.669,180.925,401.595,170.524,39.442,157.450
C08547=1041.663,180.677,401.619,170.520,39.441,157.450
C08548=1041.656,180.428,401.643,170.518,39.440,157.449
C08549=1041.651,180.179,401.666,170.515,39.439,157.449
C08550=1041.644,179.930,401.690,170.512,39.438,157.449
C08551=1041.638,179.681,401.714,170.510,39.437,157.448
C08552=1041.631,179.432,401.736,170.507,39.436,157.448
C08553=1041.625,179.184,401.760,170.505,39.435,157.448
C08554=1041.619,178.935,401.783,170.502,39.434,157.448
C08555=1041.612,178.686,401.807,170.499,39.433,157.447
C08556=1041.607,178.437,401.830,170.497,39.432,157.447
C08557=1041.600,178.188,401.854,170.494,39.431,157.447
C08558=1041.594,177.939,401.877,170.491,39.430,157.446
C08559=1041.588,177.691,401.901,170.489,39.429,157.446
C08560=1041.582,177.441,401.924,170.487,39.428,157.446
C08561=1041.576,177.193,401.948,170.483,39.427,157.446
C08562=1041.569,176.944,401.970,170.481,39.426,157.445
C08563=1041.563,176.695,401.994,170.479,39.425,157.445
C08564=1041.557,176.447,402.017,170.476,39.424,157.445
C08565=1041.550,176.198,402.041,170.473,39.423,157.444
C08566=1041.545,175.949,402.064,170.471,39.422,157.444
C08567=1041.538,175.700,402.088,170.469,39.421,157.444
C08568=1041.532,175.451,402.111,170.466,39.420,157.444
C08569=1041.526,175.203,402.135,170.463,39.419,157.443
C08570=1041.519,174.953,402.157,170.461,39.418,157.443
C08571=1041.513,174.704,402.180,170.458,39.417,157.443
C08572=1041.507,174.456,402.204,170.455,39.416,157.442
C08573=1041.501,174.207,402.227,170.453,39.415,157.442
C08574=1041.495,173.958,402.251,170.451,39.414,157.442
C08575=1041.489,173.673,402.277,170.448,39.413,157.442
C08576=1041.481,173.389,402.304,170.444,39.412,157.441
C08577=1041.474,173.103,402.331,170.442,39.411,157.441
C08578=1041.467,172.819,402.356,170.439,39.410,157.441
C08579=1041.461,172.570,402.380,170.436,39.409,157.440
C08580=1041.455,172.321,402.403,170.434,39.407,157.440
C08581=1041.449,172.072,402.426,170.431,39.406,157.440
C08582=1041.443,171.823,402.450,170.429,39.405,157.439
C08583=1041.436,171.575,402.473,170.426,39.404,157.439
C08584=1041.431,171.326,402.495,170.424,39.404,157.439
C08585=1041.425,171.077,402.519,170.421,39.403,157.439
C08586=1041.418,170.828,402.542,170.419,39.402,157.438
C08587=1041.412,170.579,402.565,170.416,39.401,157.438
C08588=1041.407,170.330,402.588,170.414,39.399,157.438
C08589=1041.401,170.081,402.611,170.411,39.398,157.437
C08590=1041.394,169.833,402.634,170.409,39.397,157.437
C08591=1041.388,169.584,402.658,170.406,39.397,157.437
C08592=1041.382,169.335,402.681,170.404,39.396,157.437
C08593=1041.376,169.086,402.704,170.401,39.395,157.436
C08594=1041.370,168.838,402.727,170.399,39.394,157.436
C08595=1041.365,168.589,402.750,170.396,39.393,157.436
C08596=1041.358,168.339,402.773,170.394,39.391,157.436
C08597=1041.352,168.090,402.796,170.392,39.390,157.435
C08598=1041.346,167.842,402.819,170.389,39.390,157.435
C08599=1041.340,167.593,402.842,170.386,39.389,157.435
C08600=1041.335,167.344,402.865,170.384,39.388,157.434
C08601=1041.328,167.096,402.888,170.382,39.387,157.434
C08602=1041.322,166.846,402.911,170.379,39.386,157.434
C08603=1041.316,166.597,402.934,170.376,39.385,157.434
C08604=1041.310,166.348,402.957,170.374,39.384,157.433
C08605=1041.304,166.100,402.980,170.372,39.383,157.433
C08606=1041.299,165.851,403.003,170.370,39.382,157.433
C08607=1041.292,165.602,403.025,170.367,39.381,157.433
C08608=1041.286,165.353,403.048,170.364,39.380,157.432
C08609=1041.281,165.104,403.071,170.362,39.379,157.432
C08610=1041.275,164.855,403.094,170.360,39.378,157.432
C08611=1041.269,164.606,403.117,170.357,39.377,157.431
C08612=1041.262,164.357,403.140,170.355,39.376,157.431
C08613=1041.256,164.108,403.163,170.353,39.375,157.431
C08614=1041.251,163.859,403.186,170.349,39.374,157.431
C08615=1041.245,163.610,403.209,170.347,39.373,157.430
C08616=1041.239,163.362,403.231,170.345,39.372,157.430
C08617=1041.233,163.113,403.254,170.343,39.371,157.430
C08618=1041.227,162.864,403.277,170.340,39.370,157.430
C08619=1041.221,162.615,403.300,170.338,39.369,157.429
C08620=1041.216,162.366,403.323,170.336,39.368,157.429
C08621=1041.209,162.118,403.345,170.333,39.367,157.429
C08622=1041.203,161.869,403.368,170.330,39.366,157.428
C08623=1041.198,161.620,403.391,170.328,39.365,157.428
C08624=1041.192,161.371,403.414,170.326,39.364,157.428
C08625=1041.186,161.122,403.437,170.324,39.363,157.428
C08626=1041.180,160.874,403.459,170.321,39.362,157.427
C08627=1041.174,160.624,403.481,170.319,39.361,157.427
C08628=1041.169,160.375,403.504,170.316,39.360,157.427
C08629=1041.163,160.126,403.527,170.314,39.359,157.427
C08630=1041.156,159.878,403.550,170.311,39.358,157.426
C08631=1041.149,159.628,403.572,170.309,39.358,157.426
C08632=1041.144,159.379,403.595,170.307,39.357,157.426
C08633=1041.137,159.130,403.617,170.305,39.356,157.425
C08634=1041.131,158.882,403.639,170.302,39.355,157.425
C08635=1041.125,158.633,403.662,170.299,39.354,157.425
C08636=1041.119,158.384,403.684,170.297,39.354,157.425
C08637=1041.113,158.135,403.707,170.295,39.353,157.425
C08638=1041.107,157.886,403.729,170.293,39.351,157.424
C08639=1041.100,157.600,403.754,170.289,39.351,157.424
C08640=1041.093,157.316,403.780,170.287,39.350,157.424
C08641=1041.086,157.030,403.805,170.284,39.349,157.423
C08642=1041.079,156.745,403.830,170.282,39.348,157.423
C08643=1041.073,156.496,403.853,170.279,39.347,157.423
C08644=1041.067,156.248,403.876,170.277,39.346,157.423
C08645=1041.061,155.998,403.898,170.274,39.345,157.422
C08646=1041.055,155.749,403.920,170.272,39.345,157.422
C08647=1041.048,155.501,403.943,170.269,39.344,157.422
C08648=1041.043,155.251,403.965,170.267,39.342,157.422
C08649=1041.037,155.003,403.987,170.265,39.342,157.422
C08650=1041.030,154.754,404.009,170.263,39.341,157.421
C08651=1041.025,154.505,404.032,170.261,39.340,157.421
C08652=1041.019,154.255,404.053,170.258,39.339,157.421
C08653=1041.012,154.007,404.076,170.255,39.339,157.421
C08654=1041.006,153.758,404.097,170.253,39.338,157.420
C08655=1041.000,153.509,404.120,170.251,39.337,157.420
C08656=1040.994,153.260,404.142,170.249,39.336,157.420
C08657=1040.988,153.011,404.164,170.246,39.335,157.420
C08658=1040.981,152.762,404.186,170.244,39.335,157.419
C08659=1040.975,152.513,404.208,170.242,39.334,157.419
C08660=1040.969,152.264,404.231,170.240,39.333,157.419
C08661=1040.963,152.015,404.253,170.236,39.332,157.419
C08662=1040.957,151.766,404.275,170.234,39.332,157.418
C08663=1040.950,151.517,404.297,170.232,39.330,157.418
C08664=1040.945,151.268,404.319,170.230,39.330,157.418
C08665=1040.938,151.019,404.342,170.228,39.329,157.418
C08666=1040.932,150.770,404.363,170.225,39.328,157.418
C08667=1040.927,150.521,404.384,170.223,39.327,157.417
C08668=1040.920,150.273,404.407,170.221,39.327,157.417
C08669=1040.915,150.023,404.429,170.219,39.326,157.417
C08670=1040.909,149.774,404.451,170.217,39.325,157.417
C08671=1040.902,149.526,404.473,170.213,39.324,157.416
C08672=1040.896,149.276,404.495,170.211,39.324,157.416
C08673=1040.890,149.028,404.517,170.209,39.323,157.416
C08674=1040.883,148.779,404.539,170.207,39.322,157.416
C08675=1040.877,148.529,404.560,170.204,39.321,157.415
C08676=1040.872,148.281,404.582,170.202,39.321,157.415
C08677=1040.866,148.032,404.604,170.200,39.319,157.415
C08678=1040.860,147.783,404.626,170.198,39.319,157.415
C08679=1040.854,147.534,404.648,170.196,39.318,157.415
C08680=1040.847,147.285,404.670,170.193,39.317,157.414
C08681=1040.841,147.036,404.692,170.191,39.316,157.414
C08682=1040.835,146.787,404.713,170.188,39.316,157.414
C08683=1040.829,146.537,404.735,170.186,39.315,157.414
C08684=1040.823,146.289,404.756,170.184,39.314,157.413
C08685=1040.817,146.040,404.779,170.182,39.314,157.413
C08686=1040.810,145.791,404.800,170.179,39.313,157.413
C08687=1040.804,145.542,404.822,170.177,39.312,157.413
C08688=1040.798,145.293,404.844,170.175,39.311,157.413
C08689=1040.792,145.043,404.865,170.173,39.311,157.412
C08690=1040.786,144.794,404.887,170.171,39.310,157.412
C08691=1040.780,144.546,404.909,170.168,39.309,157.412
C08692=1040.774,144.297,404.930,170.166,39.309,157.412
C08693=1040.768,144.048,404.952,170.164,39.307,157.411
C08694=1040.761,143.799,404.973,170.162,39.307,157.411
C08695=1040.755,143.550,404.995,170.159,39.307,157.411
C08696=1040.749,143.301,405.016,170.156,39.305,157.411
C08697=1040.743,143.052,405.038,170.154,39.305,157.411
C08698=1040.737,142.803,405.059,170.152,39.304,157.410
C08699=1040.731,142.554,405.081,170.150,39.303,157.410
C08700=1040.724,142.304,405.103,170.148,39.303,157.410
C08701=1040.718,142.057,405.125,170.145,39.302,157.410
C08702=1040.712,141.807,405.146,170.143,39.301,157.410
C08703=1040.705,141.521,405.171,170.141,39.300,157.409
C08704=1040.698,141.236,405.195,170.138,39.299,157.409
C08705=1040.691,140.950,405.220,170.135,39.299,157.409
C08706=1040.685,140.665,405.245,170.133,39.298,157.409
C08707=1040.679,140.416,405.266,170.131,39.297,157.408
C08708=1040.672,140.166,405.288,170.129,39.296,157.408
C08709=1040.665,139.917,405.309,170.127,39.295,157.408
C08710=1040.660,139.669,405.330,170.124,39.295,157.408
C08711=1040.654,139.420,405.352,170.122,39.294,157.407
C08712=1040.648,139.170,405.374,170.119,39.293,157.407
C08713=1040.642,138.922,405.395,170.117,39.293,157.407
C08714=1040.636,138.673,405.416,170.115,39.292,157.407
C08715=1040.629,138.424,405.438,170.113,39.291,157.407
C08716=1040.623,138.174,405.458,170.110,39.291,157.407
C08717=1040.618,137.926,405.480,170.108,39.290,157.406
C08718=1040.611,137.676,405.501,170.106,39.289,157.406
C08719=1040.604,137.427,405.522,170.104,39.289,157.406
C08720=1040.598,137.178,405.544,170.102,39.288,157.406
C08721=1040.593,136.930,405.565,170.099,39.287,157.405
C08722=1040.587,136.681,405.587,170.097,39.287,157.405
C08723=1040.580,136.431,405.607,170.095,39.286,157.405
C08724=1040.574,136.183,405.629,170.093,39.285,157.405
C08725=1040.568,135.933,405.650,170.091,39.285,157.405
C08726=1040.561,135.684,405.671,170.088,39.284,157.404
C08727=1040.555,135.435,405.693,170.086,39.283,157.404
C08728=1040.550,135.186,405.713,170.084,39.283,157.404
C08729=1040.543,134.937,405.734,170.082,39.281,157.404
C08730=1040.537,134.688,405.756,170.080,39.281,157.404
C08731=1040.531,134.439,405.777,170.078,39.280,157.403
C08732=1040.525,134.190,405.798,170.075,39.280,157.403
C08733=1040.519,133.941,405.819,170.073,39.279,157.403
C08734=1040.513,133.692,405.841,170.071,39.278,157.403
C08735=1040.506,133.443,405.862,170.069,39.278,157.403
C08736=1040.500,133.194,405.883,170.067,39.277,157.402
C08737=1040.495,132.945,405.904,170.064,39.276,157.402
C08738=1040.488,132.696,405.925,170.062,39.276,157.402
C08739=1040.482,132.446,405.946,170.060,39.275,157.402
C08740=1040.476,132.198,405.967,170.058,39.274,157.402
C08741=1040.469,131.949,405.988,170.056,39.274,157.401
C08742=1040.464,131.700,406.009,170.054,39.273,157.401
C08743=1040.458,131.451,406.030,170.051,39.272,157.401
C08744=1040.451,131.202,406.051,170.049,39.272,157.401
C08745=1040.446,130.953,406.072,170.047,39.271,157.401
C08746=1040.439,130.704,406.093,170.045,39.270,157.400
C08747=1040.433,130.454,406.114,170.043,39.270,157.400
C08748=1040.427,130.206,406.134,170.041,39.269,157.400
C08749=1040.420,129.956,406.155,170.038,39.269,157.400
C08750=1040.414,129.707,406.176,170.036,39.268,157.400
C08751=1040.408,129.458,406.196,170.034,39.268,157.400
C08752=1040.401,129.209,406.217,170.032,39.267,157.399
C08753=1040.395,128.960,406.239,170.030,39.266,157.399
C08754=1040.389,128.711,406.259,170.028,39.266,157.399
C08755=1040.382,128.462,406.279,170.025,39.265,157.399
C08756=1040.376,128.212,406.301,170.023,39.265,157.399
C08757=1040.370,127.964,406.321,170.021,39.264,157.398
C08758=1040.363,127.715,406.342,170.019,39.264,157.398
C08759=1040.358,127.466,406.363,170.017,39.262,157.398
C08760=1040.351,127.217,406.384,170.015,39.262,157.398
C08761=1040.345,126.967,406.404,170.012,39.261,157.398
C08762=1040.339,126.719,406.425,170.010,39.261,157.398
C08763=1040.332,126.469,406.446,170.008,39.261,157.397
C08764=1040.326,126.221,406.466,170.006,39.260,157.397
C08765=1040.320,125.971,406.487,170.004,39.259,157.397
C08766=1040.314,125.722,406.507,170.002,39.258,157.397
C08767=1040.307,125.436,406.531,169.998,39.258,157.397
C08768=1040.300,125.151,406.555,169.996,39.258,157.396
C08769=1040.292,124.865,406.579,169.994,39.256,157.396
C08770=1040.285,124.579,406.602,169.991,39.256,157.396
C08771=1040.279,124.330,406.623,169.989,39.256,157.396
C08772=1040.273,124.081,406.643,169.987,39.255,157.396
C08773=1040.267,123.831,406.664,169.984,39.254,157.395
C08774=1040.261,123.583,406.685,169.983,39.253,157.395
C08775=1040.254,123.333,406.705,169.981,39.253,157.395
C08776=1040.248,123.084,406.725,169.979,39.252,157.395
C08777=1040.242,122.835,406.747,169.977,39.252,157.395
C08778=1040.236,122.586,406.767,169.974,39.251,157.394
C08779=1040.230,122.337,406.787,169.972,39.250,157.394
C08780=1040.223,122.089,406.808,169.970,39.250,157.394
C08781=1040.218,121.839,406.829,169.968,39.249,157.394
C08782=1040.212,121.590,406.849,169.966,39.249,157.394
C08783=1040.205,121.341,406.869,169.964,39.248,157.394
C08784=1040.199,121.092,406.890,169.962,39.247,157.393
C08785=1040.193,120.843,406.911,169.959,39.247,157.393
C08786=1040.187,120.594,406.931,169.957,39.246,157.393
C08787=1040.181,120.344,406.951,169.955,39.246,157.393
C08788=1040.175,120.096,406.972,169.953,39.245,157.393
C08789=1040.169,119.847,406.992,169.951,39.244,157.392
C08790=1040.162,119.597,407.012,169.949,39.244,157.392
C08791=1040.157,119.348,407.033,169.946,39.243,157.392
C08792=1040.150,119.099,407.054,169.944,39.243,157.392
C08793=1040.144,118.851,407.074,169.942,39.242,157.392
C08794=1040.138,118.601,407.095,169.940,39.241,157.391
C08795=1040.132,118.352,407.115,169.938,39.241,157.391
C08796=1040.125,118.102,407.135,169.937,39.240,157.391
C08797=1040.120,117.854,407.155,169.934,39.240,157.391
C08798=1040.114,117.605,407.176,169.932,39.239,157.391
C08799=1040.107,117.356,407.197,169.930,39.238,157.391
C08800=1040.101,117.107,407.217,169.928,39.237,157.390
C08801=1040.095,116.857,407.238,169.926,39.237,157.390
C08802=1040.089,116.608,407.258,169.924,39.236,157.390
C08803=1040.084,116.359,407.278,169.921,39.236,157.390
C08804=1040.077,116.110,407.298,169.919,39.235,157.390
C08805=1040.072,115.861,407.318,169.917,39.234,157.389
C08806=1040.066,115.612,407.338,169.915,39.234,157.389
C08807=1040.059,115.363,407.359,169.913,39.233,157.389
C08808=1040.053,115.114,407.379,169.910,39.232,157.389
C08809=1040.047,114.864,407.400,169.909,39.232,157.389
C08810=1040.041,114.615,407.420,169.907,39.231,157.389
C08811=1040.035,114.367,407.440,169.905,39.231,157.388
C08812=1040.028,114.117,407.461,169.903,39.230,157.388
C08813=1040.023,113.868,407.481,169.901,39.229,157.388
C08814=1040.017,113.619,407.501,169.899,39.229,157.388
C08815=1040.010,113.370,407.521,169.896,39.228,157.388
C08816=1040.004,113.121,407.541,169.894,39.228,157.387
C08817=1039.998,112.872,407.561,169.892,39.227,157.387
C08818=1039.992,112.623,407.582,169.890,39.227,157.387
C08819=1039.986,112.374,407.602,169.888,39.226,157.387
C08820=1039.980,112.125,407.622,169.886,39.225,157.387
C08821=1039.974,111.875,407.641,169.883,39.225,157.387
C08822=1039.968,111.626,407.661,169.882,39.224,157.386
C08823=1039.962,111.377,407.681,169.880,39.223,157.386
C08824=1039.955,111.128,407.701,169.878,39.223,157.386
C08825=1039.949,110.879,407.721,169.876,39.222,157.386
C08826=1039.942,110.629,407.742,169.874,39.222,157.386
C08827=1039.936,110.381,407.762,169.872,39.222,157.386
C08828=1039.930,110.132,407.782,169.869,39.221,157.385
C08829=1039.924,109.882,407.801,169.867,39.221,157.385
C08830=1039.918,109.633,407.821,169.865,39.220,157.385
C08831=1039.911,109.347,407.843,169.863,39.220,157.385
C08832=1039.904,109.061,407.866,169.861,39.218,157.385
C08833=1039.896,108.775,407.889,169.858,39.218,157.385
C08834=1039.889,108.489,407.912,169.855,39.217,157.384
C08835=1039.883,108.240,407.932,169.853,39.217,157.384
C08836=1039.877,107.991,407.951,169.851,39.217,157.384
C08837=1039.870,107.742,407.972,169.849,39.216,157.384
C08838=1039.864,107.492,407.991,169.847,39.216,157.384
C08839=1039.858,107.244,408.011,169.845,39.215,157.384
C08840=1039.852,106.994,408.031,169.844,39.214,157.383
C08841=1039.846,106.745,408.051,169.841,39.214,157.383
C08842=1039.839,106.496,408.070,169.839,39.213,157.383
C08843=1039.833,106.247,408.090,169.837,39.213,157.383
C08844=1039.827,105.998,408.110,169.835,39.213,157.383
C08845=1039.821,105.748,408.129,169.833,39.212,157.383
C08846=1039.815,105.500,408.149,169.831,39.212,157.382
C08847=1039.808,105.250,408.169,169.828,39.210,157.382
C08848=1039.802,105.001,408.188,169.826,39.210,157.382
C08849=1039.796,104.752,408.208,169.824,39.209,157.382
C08850=1039.790,104.503,408.228,169.822,39.209,157.382
C08851=1039.784,104.253,408.248,169.820,39.208,157.382
C08852=1039.778,104.004,408.268,169.819,39.208,157.381
C08853=1039.771,103.756,408.287,169.817,39.207,157.381
C08854=1039.765,103.506,408.306,169.815,39.207,157.381
C08855=1039.759,103.258,408.326,169.812,39.206,157.381
C08856=1039.753,103.008,408.347,169.810,39.206,157.381
C08857=1039.747,102.759,408.366,169.808,39.205,157.381
C08858=1039.740,102.510,408.385,169.806,39.205,157.380
C08859=1039.735,102.261,408.405,169.804,39.204,157.380
C08860=1039.728,102.011,408.425,169.802,39.204,157.380
C08861=1039.722,101.762,408.444,169.800,39.203,157.380
C08862=1039.716,101.513,408.464,169.798,39.203,157.380
C08863=1039.710,101.264,408.483,169.796,39.202,157.379
C08864=1039.704,101.015,408.503,169.794,39.201,157.379
C08865=1039.698,100.766,408.523,169.792,39.201,157.379
C08866=1039.692,100.516,408.542,169.790,39.200,157.379
C08867=1039.685,100.268,408.562,169.788,39.200,157.379
C08868=1039.679,100.018,408.581,169.785,39.199,157.379
C08869=1039.673,99.769,408.601,169.783,39.199,157.379
C08870=1039.666,99.519,408.620,169.781,39.198,157.378
C08871=1039.660,99.271,408.640,169.779,39.198,157.378
C08872=1039.654,99.022,408.658,169.778,39.197,157.378
C08873=1039.648,98.772,408.678,169.776,39.197,157.378
C08874=1039.641,98.524,408.697,169.774,39.197,157.378
C08875=1039.635,98.273,408.717,169.772,39.196,157.378
C08876=1039.628,98.025,408.736,169.769,39.196,157.378
C08877=1039.623,97.776,408.755,169.767,39.195,157.377
C08878=1039.616,97.526,408.774,169.765,39.195,157.377
C08879=1039.610,97.278,408.794,169.763,39.194,157.377
C08880=1039.604,97.028,408.813,169.761,39.194,157.377
C08881=1039.597,96.778,408.832,169.759,39.193,157.377
C08882=1039.592,96.530,408.852,169.757,39.193,157.377
C08883=1039.585,96.280,408.871,169.754,39.192,157.376
C08884=1039.579,96.032,408.891,169.753,39.192,157.376
C08885=1039.573,95.782,408.909,169.751,39.191,157.376
C08886=1039.567,95.533,408.929,169.749,39.191,157.376
C08887=1039.561,95.284,408.947,169.747,39.190,157.376
C08888=1039.554,95.034,408.968,169.745,39.190,157.376
C08889=1039.548,94.785,408.986,169.743,39.189,157.376
C08890=1039.542,94.536,409.005,169.740,39.189,157.375
C08891=1039.535,94.287,409.025,169.738,39.188,157.375
C08892=1039.529,94.038,409.044,169.736,39.188,157.375
C08893=1039.523,93.789,409.063,169.735,39.187,157.375
C08894=1039.517,93.540,409.083,169.733,39.187,157.375
C08895=1039.510,93.254,409.104,169.730,39.186,157.375
C08896=1039.503,92.967,409.126,169.728,39.186,157.374
C08897=1039.495,92.682,409.148,169.725,39.185,157.374
C08898=1039.488,92.395,409.170,169.723,39.185,157.374
C08899=1039.482,92.146,409.190,169.721,39.184,157.374
C08900=1039.476,91.897,409.208,169.719,39.184,157.374
C08901=1039.470,91.648,409.228,169.717,39.183,157.374
C08902=1039.464,91.399,409.246,169.715,39.183,157.373
C08903=1039.458,91.149,409.266,169.714,39.182,157.373
C08904=1039.451,90.901,409.285,169.712,39.182,157.373
C08905=1039.446,90.651,409.304,169.709,39.181,157.373
C08906=1039.439,90.402,409.323,169.707,39.181,157.373
C08907=1039.433,90.153,409.342,169.705,39.180,157.373
C08908=1039.427,89.904,409.361,169.703,39.180,157.372
C08909=1039.420,89.654,409.380,169.701,39.179,157.372
C08910=1039.414,89.404,409.399,169.699,39.179,157.372
C08911=1039.408,89.155,409.418,169.697,39.178,157.372
C08912=1039.401,88.907,409.437,169.694,39.178,157.372
C08913=1039.395,88.658,409.456,169.693,39.177,157.372
C08914=1039.388,88.409,409.474,169.691,39.177,157.372
C08915=1039.383,88.159,409.494,169.689,39.177,157.372
C08916=1039.376,87.910,409.512,169.687,39.176,157.371
C08917=1039.370,87.661,409.531,169.685,39.176,157.371
C08918=1039.363,87.412,409.550,169.683,39.175,157.371
C08919=1039.358,87.162,409.569,169.681,39.175,157.371
C08920=1039.351,86.913,409.587,169.678,39.174,157.371
C08921=1039.345,86.664,409.606,169.676,39.174,157.371
C08922=1039.338,86.415,409.625,169.674,39.173,157.370
C08923=1039.332,86.166,409.643,169.672,39.174,157.370
C08924=1039.326,85.916,409.663,169.671,39.173,157.370
C08925=1039.320,85.667,409.681,169.669,39.173,157.370
C08926=1039.313,85.418,409.700,169.667,39.172,157.370
C08927=1039.307,85.169,409.719,169.665,39.172,157.370
C08928=1039.300,84.920,409.737,169.662,39.171,157.370
C08929=1039.295,84.671,409.756,169.660,39.171,157.369
C08930=1039.289,84.421,409.774,169.658,39.170,157.369
C08931=1039.282,84.172,409.793,169.656,39.170,157.369
C08932=1039.276,83.923,409.812,169.654,39.169,157.369
C08933=1039.269,83.673,409.830,169.653,39.169,157.369
C08934=1039.264,83.424,409.850,169.651,39.169,157.369
C08935=1039.257,83.175,409.868,169.649,39.168,157.369
C08936=1039.251,82.926,409.887,169.646,39.168,157.368
C08937=1039.244,82.677,409.906,169.644,39.167,157.368
C08938=1039.238,82.428,409.924,169.642,39.167,157.368
C08939=1039.232,82.178,409.943,169.640,39.166,157.368
C08940=1039.226,81.928,409.961,169.638,39.166,157.368
C08941=1039.220,81.679,409.980,169.636,39.165,157.368
C08942=1039.213,81.430,409.999,169.635,39.165,157.368
C08943=1039.207,81.181,410.017,169.632,39.164,157.367
C08944=1039.201,80.932,410.037,169.630,39.164,157.367
C08945=1039.195,80.682,410.055,169.628,39.163,157.367
C08946=1039.188,80.433,410.074,169.626,39.163,157.367
C08947=1039.182,80.184,410.092,169.624,39.163,157.367
C08948=1039.176,79.935,410.110,169.622,39.162,157.367
C08949=1039.170,79.686,410.129,169.620,39.162,157.367
C08950=1039.164,79.437,410.148,169.619,39.161,157.366
C08951=1039.158,79.187,410.167,169.616,39.161,157.366
C08952=1039.152,78.938,410.185,169.614,39.160,157.366
C08953=1039.145,78.689,410.203,169.612,39.160,157.366
C08954=1039.139,78.440,410.222,169.610,39.159,157.366
C08955=1039.133,78.190,410.240,169.608,39.159,157.366
C08956=1039.126,77.941,410.258,169.606,39.158,157.365
C08957=1039.120,77.692,410.277,169.604,39.158,157.365
C08958=1039.114,77.443,410.295,169.602,39.158,157.365
C08959=1039.107,77.157,410.317,169.599,39.157,157.365
C08960=1039.100,76.870,410.338,169.597,39.157,157.365
C08961=1039.093,76.585,410.359,169.595,39.156,157.365
C08962=1039.086,76.298,410.380,169.593,39.156,157.365
C08963=1039.079,76.049,410.398,169.591,39.155,157.364
C08964=1039.072,75.800,410.416,169.589,39.155,157.364
C08965=1039.066,75.551,410.435,169.587,39.154,157.364
C08966=1039.060,75.301,410.453,169.585,39.154,157.364
C08967=1039.054,75.052,410.471,169.582,39.153,157.364
C08968=1039.048,74.803,410.490,169.580,39.153,157.364
C08969=1039.042,74.553,410.508,169.578,39.153,157.364
C08970=1039.035,74.304,410.526,169.577,39.152,157.363
C08971=1039.029,74.055,410.544,169.575,39.152,157.363
C08972=1039.023,73.805,410.563,169.573,39.151,157.363
C08973=1039.016,73.556,410.581,169.571,39.151,157.363
C08974=1039.010,73.308,410.598,169.569,39.151,157.363
C08975=1039.003,73.059,410.617,169.567,39.151,157.363
C08976=1038.997,72.809,410.635,169.564,39.150,157.363
C08977=1038.991,72.560,410.654,169.562,39.150,157.362
C08978=1038.985,72.310,410.672,169.560,39.149,157.362
C08979=1038.978,72.061,410.690,169.559,39.148,157.362
C08980=1038.973,71.812,410.708,169.557,39.149,157.362
C08981=1038.966,71.563,410.726,169.555,39.148,157.362
C08982=1038.960,71.313,410.744,169.553,39.148,157.362
C08983=1038.953,71.064,410.762,169.551,39.147,157.362
C08984=1038.947,70.814,410.780,169.548,39.147,157.362
C08985=1038.941,70.566,410.799,169.546,39.146,157.361
C08986=1038.935,70.316,410.817,169.544,39.146,157.361
C08987=1038.929,70.067,410.835,169.542,39.146,157.361
C08988=1038.923,69.817,410.853,169.541,39.145,157.361
C08989=1038.916,69.568,410.871,169.539,39.145,157.361
C08990=1038.910,69.319,410.889,169.537,39.144,157.361
C08991=1038.904,69.070,410.907,169.535,39.144,157.361
C08992=1038.897,68.821,410.925,169.532,39.143,157.360
C08993=1038.891,68.571,410.943,169.530,39.143,157.360
C08994=1038.884,68.321,410.961,169.528,39.143,157.360
C08995=1038.879,68.073,410.979,169.526,39.142,157.360
C08996=1038.872,67.823,410.997,169.524,39.142,157.360
C08997=1038.866,67.574,411.015,169.522,39.141,157.360
C08998=1038.859,67.325,411.033,169.520,39.141,157.360
C08999=1038.854,67.076,411.050,169.519,39.141,157.360
C09000=1038.847,66.827,411.069,169.517,39.140,157.359
C09001=1038.840,66.577,411.086,169.514,39.140,157.359
C09002=1038.834,66.327,411.104,169.512,39.139,157.359
C09003=1038.829,66.078,411.122,169.510,39.139,157.359
C09004=1038.822,65.830,411.140,169.508,39.139,157.359
C09005=1038.815,65.580,411.158,169.506,39.138,157.359
C09006=1038.809,65.330,411.176,169.504,39.138,157.359
C09007=1038.803,65.082,411.194,169.502,39.138,157.359
C09008=1038.797,64.832,411.211,169.500,39.138,157.358
C09009=1038.790,64.582,411.229,169.499,39.137,157.358
C09010=1038.784,64.333,411.247,169.496,39.137,157.358
C09011=1038.778,64.085,411.265,169.494,39.136,157.358
C09012=1038.772,63.835,411.283,169.492,39.136,157.358
C09013=1038.765,63.585,411.300,169.490,39.136,157.358
C09014=1038.759,63.336,411.318,169.488,39.135,157.358
C09015=1038.752,63.087,411.335,169.486,39.135,157.358
C09016=1038.746,62.837,411.353,169.484,39.135,157.357
C09017=1038.739,62.588,411.371,169.482,39.134,157.357
C09018=1038.732,62.339,411.389,169.480,39.134,157.357
C09019=1038.727,62.090,411.406,169.478,39.134,157.357
C09020=1038.720,61.841,411.423,169.475,39.133,157.357
C09021=1038.714,61.591,411.441,169.473,39.134,157.357
C09022=1038.707,61.341,411.459,169.471,39.133,157.357
C09023=1038.700,61.055,411.479,169.469,39.133,157.357
C09024=1038.692,60.769,411.499,169.467,39.132,157.356
C09025=1038.685,60.483,411.519,169.465,39.132,157.356
C09026=1038.677,60.197,411.539,169.463,39.132,157.356
C09027=1038.672,59.947,411.556,169.461,39.131,157.356
C09028=1038.665,59.698,411.574,169.459,39.131,157.356
C09029=1038.659,59.448,411.591,169.457,39.131,157.356
C09030=1038.652,59.200,411.608,169.454,39.130,157.356
C09031=1038.645,58.951,411.627,169.452,39.130,157.356
C09032=1038.639,58.701,411.644,169.450,39.130,157.355
C09033=1038.633,58.452,411.661,169.448,39.129,157.355
C09034=1038.627,58.203,411.679,169.446,39.130,157.355
C09035=1038.620,57.953,411.697,169.444,39.129,157.355
C09036=1038.614,57.704,411.714,169.442,39.129,157.355
C09037=1038.607,57.455,411.732,169.440,39.128,157.355
C09038=1038.601,57.205,411.749,169.438,39.128,157.355
C09039=1038.594,56.956,411.766,169.436,39.128,157.355
C09040=1038.589,56.706,411.783,169.433,39.127,157.354
C09041=1038.582,56.457,411.800,169.432,39.127,157.354
C09042=1038.575,56.208,411.817,169.430,39.127,157.354
C09043=1038.569,55.958,411.835,169.428,39.126,157.354
C09044=1038.562,55.709,411.853,169.426,39.126,157.354
C09045=1038.557,55.460,411.870,169.424,39.126,157.354
C09046=1038.550,55.210,411.888,169.422,39.125,157.354
C09047=1038.544,54.962,411.905,169.420,39.125,157.354
C09048=1038.538,54.712,411.923,169.418,39.125,157.354
C09049=1038.531,54.462,411.940,169.416,39.125,157.353
C09050=1038.525,54.214,411.957,169.413,39.124,157.353
C09051=1038.518,53.964,411.975,169.411,39.124,157.353
C09052=1038.512,53.715,411.992,169.409,39.124,157.353
C09053=1038.506,53.465,412.008,169.407,39.123,157.353
C09054=1038.500,53.216,412.026,169.405,39.123,157.353
C09055=1038.493,52.967,412.043,169.404,39.123,157.353
C09056=1038.486,52.717,412.061,169.402,39.122,157.353
C09057=1038.481,52.468,412.078,169.400,39.122,157.352
C09058=1038.474,52.219,412.095,169.398,39.121,157.352
C09059=1038.468,51.970,412.112,169.395,39.121,157.352
C09060=1038.462,51.720,412.130,169.393,39.121,157.352
C09061=1038.456,51.471,412.147,169.391,39.120,157.352
C09062=1038.449,51.222,412.164,169.389,39.120,157.352
C09063=1038.443,50.973,412.182,169.387,39.120,157.352
C09064=1038.437,50.723,412.199,169.385,39.119,157.352
C09065=1038.431,50.474,412.215,169.383,39.119,157.351
C09066=1038.424,50.224,412.233,169.381,39.119,157.351
C09067=1038.418,49.975,412.250,169.379,39.119,157.351
C09068=1038.411,49.726,412.267,169.378,39.118,157.351
C09069=1038.406,49.475,412.285,169.375,39.118,157.351
C09070=1038.399,49.227,412.302,169.373,39.118,157.351
C09071=1038.393,48.978,412.319,169.371,39.117,157.351
C09072=1038.387,48.728,412.336,169.369,39.117,157.351
C09073=1038.381,48.479,412.353,169.367,39.116,157.350
C09074=1038.374,48.230,412.370,169.365,39.116,157.350
C09075=1038.369,47.980,412.388,169.363,39.116,157.350
C09076=1038.362,47.731,412.405,169.361,39.115,157.350
C09077=1038.356,47.482,412.421,169.359,39.115,157.350
C09078=1038.350,47.232,412.439,169.356,39.114,157.350
C09079=1038.343,46.983,412.456,169.354,39.114,157.350
C09080=1038.337,46.733,412.473,169.352,39.114,157.350
C09081=1038.331,46.484,412.490,169.351,39.113,157.349
C09082=1038.324,46.235,412.508,169.349,39.113,157.349
C09083=1038.318,45.985,412.524,169.347,39.112,157.349
C09084=1038.312,45.737,412.541,169.345,39.112,157.349
C09085=1038.306,45.487,412.559,169.343,39.112,157.349
C09086=1038.300,45.238,412.575,169.341,39.111,157.349
C09087=1038.293,44.951,412.595,169.338,39.111,157.349
C09088=1038.286,44.664,412.615,169.336,39.110,157.348
C09089=1038.279,44.378,412.634,169.333,39.110,157.348
C09090=1038.271,44.091,412.654,169.331,39.109,157.348
C09091=1038.266,43.842,412.670,169.329,39.110,157.348
C09092=1038.259,43.592,412.688,169.327,39.109,157.348
C09093=1038.253,43.343,412.704,169.325,39.109,157.348
C09094=1038.247,43.094,412.722,169.323,39.108,157.348
C09095=1038.241,42.845,412.739,169.321,39.108,157.348
C09096=1038.235,42.595,412.755,169.319,39.108,157.347
C09097=1038.228,42.346,412.773,169.317,39.107,157.347
C09098=1038.222,42.096,412.789,169.315,39.107,157.347
C09099=1038.215,41.846,412.805,169.313,39.107,157.347
C09100=1038.209,41.598,412.822,169.311,39.106,157.347
C09101=1038.203,41.348,412.839,169.309,39.106,157.347
C09102=1038.196,41.099,412.856,169.307,39.106,157.347
